(* IEC 61131-3 sources: Industry-PLC-LLM/data/PLCBEAD_repo/PLCBEAD_PLCEmbed-main/PLC-BEAD/Source/OpenPLCv2 (part 9) *)

(* ---- SRAMP.ST ---- *)
FUNCTION_BLOCK T_PLC_US_Block
	VAR_OUTPUT
		T_PLC_US :	UDINT;
	END_VAR

	VAR_EXTERNAL
		PLC_TICKS_PER_SEC :	INT;
		PLC_SYS_TICK_CNT :	DINT;
	END_VAR

	VAR
		debug :	BOOL;
		N :	INT;
		Offset :	UDINT;
		temp :	DWORD := DWORD#1;
		mode :	BOOL;
		faktor :	UDINT;
		init :	BOOL;
		v_plc_ticks_per_sec :	UDINT;
		base :	UDINT := UDINT#1000000;
	END_VAR

	IF init = FALSE THEN
		v_plc_ticks_per_sec := INT_TO_UDINT(PLC_TICKS_PER_SEC);
		IF v_plc_ticks_per_sec = UDINT#1024 THEN
			faktor := UDINT#1000;
			mode := FALSE;
		ELSIF v_plc_ticks_per_sec > UDINT#0 THEN
			IF v_plc_ticks_per_sec <= base THEN
				faktor := base / v_plc_ticks_per_sec;
				mode := FALSE;
			ELSE
				faktor := v_plc_ticks_per_sec / base;
				mode := TRUE;
			END_IF;
		ELSE
			faktor := UDINT#1;
		END_IF;
		init := TRUE;
	END_IF;

	IF mode THEN
		T_PLC_US := DINT_TO_UDINT(PLC_SYS_TICK_CNT) / faktor;
	ELSE
		T_PLC_US := DINT_TO_UDINT(PLC_SYS_TICK_CNT) * faktor;
	END_IF;

	IF debug THEN
		T_PLC_US := (DWORD_TO_UDINT(SHL(UDINT_TO_DWORD(T_PLC_US),N) OR SHL(temp,N)) - UDINT#1) + Offset;
	END_IF;
END_FUNCTION_BLOCK

FUNCTION_BLOCK TC_S_Block

	VAR_OUTPUT
		TC :	REAL;
	END_VAR

	VAR
		init :	BOOL;
		tx :	UDINT;
		last :	UDINT;
		T_PLC_US :	T_PLC_US_Block;
	END_VAR

	T_PLC_US();
	tx:= T_PLC_US.T_PLC_US;

	IF NOT init THEN
		init := TRUE;
		TC := 0.0;
	ELSE
		tc := UDINT_TO_REAL(tx - last) * 1.0E-6;
	END_IF;
	last := tx;

END_FUNCTION_BLOCK

FUNCTION_BLOCK SRAMP_Block

	VAR_INPUT
		X :	REAL;
		A_UP :	REAL;
		A_DN :	REAL;
		VU_MAX :	REAL;
		VD_MAX :	REAL;
		LIMIT_HIGH :	REAL;
		LIMIT_LOW :	REAL;
		RST :	BOOL;
	END_VAR

	VAR_OUTPUT
		Y :	REAL;
		V :	REAL;
	END_VAR

	VAR
		cycle_time :	TC_S_Block;
		init :	BOOL;
	END_VAR

	cycle_time();

	A_up := MAX(0.0,A_UP);
	A_dn := MIN(0.0,A_dn);
	VU_max := MAX(0.0,VU_max);
	VD_max := MIN(0.0,VD_MAX);

	IF rst OR NOT init THEN
		init := TRUE;
		Y := 0.0;
		V := 0.0;
	ELSIF X = Y THEN
		v := 0.0;
	ELSIF X > Y THEN
		v := MIN(v + A_UP * cycle_time.TC, vu_max);
		v := MIN(SQRT((Y-X) * 2.0 * A_DN), v);
		y := LIMIT(limit_low, y + MIN(v * cycle_time.TC, X-Y), limit_high);
	ELSIF X < Y THEN
		v := MAX(v + A_DN * cycle_time.TC, vd_max);
		v := MAX(-SQRT((Y-X) * 2.0 * A_UP), v);
		y := LIMIT(limit_low, y + MAX(v * cycle_time.TC, X-Y), limit_high);
	END_IF;

END_FUNCTION_BLOCK

PROGRAM program0
	VAR
		X :	REAL;
		A_UP :	REAL;
		A_DN :	REAL;
		VU_MAX :	REAL;
		VD_MAX :	REAL;
		LIMIT_HIGH :	REAL;
		LIMIT_LOW :	REAL;
		RST :	BOOL;
		Y :	REAL;
		V :	REAL;
		func_block : SRAMP_Block;
	END_VAR
		func_block.X  := X;
		func_block.A_UP  := A_UP;
		func_block.A_DN  := A_DN;
		func_block.VU_MAX  := VU_MAX;
		func_block.VD_MAX  := VD_MAX;
		func_block.LIMIT_HIGH  := LIMIT_HIGH;
		func_block.LIMIT_LOW  := LIMIT_LOW;
		func_block.RST  := RST;
		func_block();
		Y := func_block.Y;
		V := func_block.V;

END_PROGRAM

CONFIGURATION Config0

	VAR_GLOBAL
		PLC_TICKS_PER_SEC :	INT;
		PLC_SYS_TICK_CNT :	DINT;
	END_VAR

	RESOURCE Res0 ON PLC
		TASK task0(INTERVAL := T#20ms,PRIORITY := 0);
		PROGRAM instance0 WITH task0 : program0;
	END_RESOURCE

END_CONFIGURATION

(* ---- STACK_16.ST ---- *)
TYPE
  oscat_ardw_0_15             : ARRAY [0..15]   OF DWORD;
END_TYPE

FUNCTION_BLOCK STACK_16_Block

	VAR_INPUT
		DIN :	DWORD;
		E :	BOOL := TRUE;
		RD :	BOOL;
		WD :	BOOL;
		RST :	BOOL;
	END_VAR

	VAR_OUTPUT
		DOUT :	DWORD;
		EMPTY :	BOOL := TRUE;
		FULL :	BOOL;
	END_VAR

	VAR
		pt :	INT;
		stack :	oscat_ardw_0_15;
	END_VAR

	IF RST THEN
		pt := 0;
		EMPTY := TRUE;
		FULL := FALSE;
		Dout := DWORD#0;
	ELSIF E THEN
		IF NOT EMPTY AND RD THEN
			pt := pt - 1;
			Dout := stack[pt];
			EMPTY := pt = 0;
			FULL := FALSE;
		END_IF;
		IF NOT FULL AND WD THEN
			stack[pt] := Din;
			pt := pt + 1;
			FULL := pt > 15;
			EMPTY := FALSE;
		END_IF;
	END_IF;

END_FUNCTION_BLOCK

PROGRAM program0
	VAR
		DIN :	DWORD;
		E :	BOOL := TRUE;
		RD :	BOOL;
		WD :	BOOL;
		RST :	BOOL;
		DOUT :	DWORD;
		EMPTY :	BOOL := TRUE;
		FULL :	BOOL;
		func_block : STACK_16_Block;
	END_VAR
		func_block.DIN  := DIN;
		func_block.E  := E;
		func_block.RD  := RD;
		func_block.WD  := WD;
		func_block.RST  := RST;
		func_block();
		DOUT := func_block.DOUT;
		EMPTY := func_block.EMPTY;
		FULL := func_block.FULL;

END_PROGRAM

CONFIGURATION Config0

	RESOURCE Res0 ON PLC
		TASK task0(INTERVAL := T#20ms,PRIORITY := 0);
		PROGRAM instance0 WITH task0 : program0;
	END_RESOURCE

END_CONFIGURATION

(* ---- STACK_32.ST ---- *)
TYPE
  	oscat_ardw_0_31             : ARRAY [0..31]   OF DWORD;
END_TYPE

FUNCTION_BLOCK STACK_32_Block

	VAR_INPUT
		DIN :	DWORD;
		E :	BOOL := TRUE;
		RD :	BOOL;
		WD :	BOOL;
		RST :	BOOL;
	END_VAR

	VAR_OUTPUT
		DOUT :	DWORD;
		EMPTY :	BOOL := TRUE;
		FULL :	BOOL;
	END_VAR

	VAR
		pt :	INT;
		stack :	oscat_ardw_0_31;
	END_VAR

	IF RST THEN
		pt := 0;
		EMPTY := TRUE;
		FULL := FALSE;
		Dout := DWORD#0;
	ELSIF E THEN
		IF NOT EMPTY AND RD THEN
			(* read one element *)
			pt := pt - 1;
			Dout := stack[pt];
			EMPTY := pt = 0;
			FULL := FALSE;
		END_IF;
		IF NOT FULL AND WD THEN
			(* write one element *)
			stack[pt] := Din;
			pt := pt + 1;
			FULL := pt > 31;
			EMPTY := FALSE;
		END_IF;
	END_IF;

END_FUNCTION_BLOCK

PROGRAM program0
	VAR
		DIN :	DWORD;
		E :	BOOL := TRUE;
		RD :	BOOL;
		WD :	BOOL;
		RST :	BOOL;
		DOUT :	DWORD;
		EMPTY :	BOOL := TRUE;
		FULL :	BOOL;
		func_block : STACK_32_Block;
	END_VAR
		func_block.DIN  := DIN;
		func_block.E  := E;
		func_block.RD  := RD;
		func_block.WD  := WD;
		func_block.RST  := RST;
		func_block();
		DOUT := func_block.DOUT;
		EMPTY := func_block.EMPTY;
		FULL := func_block.FULL;

END_PROGRAM

CONFIGURATION Config0

	RESOURCE Res0 ON PLC
		TASK task0(INTERVAL := T#20ms,PRIORITY := 0);
		PROGRAM instance0 WITH task0 : program0;
	END_RESOURCE

END_CONFIGURATION

(* ---- STAIR2.ST ---- *)
FUNCTION FLOOR : INT
	VAR_INPUT
		x : REAL;
	END_VAR

	FLOOR := REAL_TO_INT(X);
	IF INT_TO_REAL(FLOOR) > X THEN
		floor := floor - 1;
	END_IF;
END_FUNCTION

FUNCTION_BLOCK STAIR2_Block

	VAR_INPUT
		X :	REAL;
		D :	REAL;
	END_VAR

	VAR_OUTPUT
		Y :	REAL;
	END_VAR

	IF D > 0.0 THEN
		IF X >= Y + D OR X <= Y - D THEN Y := INT_TO_REAL(FLOOR(X/D)) * D; END_IF;
	ELSE
		Y := X;
	END_IF;

END_FUNCTION_BLOCK

PROGRAM program0

	VAR
		X :	REAL;
		D :	REAL;
		Y :	REAL;
		func_block : STAIR2_Block;
	END_VAR
	func_block.X := X;
	func_block.D := D;
	func_block();
	Y := func_block.Y;

END_PROGRAM

CONFIGURATION Config0

	RESOURCE Res0 ON PLC
		TASK task0(INTERVAL := T#20ms,PRIORITY := 0);
		PROGRAM instance0 WITH task0 : program0;
	END_RESOURCE

END_CONFIGURATION

(* ---- STATUS_TO_ESR.ST ---- *)
TYPE
  oscat_esr_collect_data      : ARRAY [0..7]    OF BYTE;
END_TYPE

TYPE oscat_esr_data :
  STRUCT
	typ    : BYTE;
	adress : STRING;
	DS     : UDINT;
	TS     : TIME;
	data   : oscat_esr_collect_data;
  END_STRUCT;
END_TYPE

FUNCTION_BLOCK STATUS_TO_ESR_Block

	VAR_INPUT
		STATUS :	BYTE;
		ADRESS :	STRING;
		DT_IN :	UDINT;
		TS :	TIME;
	END_VAR

	VAR_OUTPUT
		STATUS_TO_ESR :	oscat_esr_data;
	END_VAR

	IF status < BYTE#100 THEN
		status_to_ESR.typ := BYTE#1;
	ELSIF status < BYTE#200 THEN
		status_to_ESR.typ := BYTE#2;
	ELSE
		status_to_ESR.typ := BYTE#3;
	END_IF;
	status_to_ESR.adress:= adress;
	status_to_ESR.DS := DT_in;
	status_to_ESR.TS := TS;
	status_to_ESR.data[0] := status;
END_FUNCTION_BLOCK

PROGRAM program0
	VAR
		STATUS :	BYTE;
		ADRESS :	STRING;
		DT_IN  :	UDINT;
		TS     :	TIME;
		STATUS_TO_ESR :	oscat_esr_data;

		func_block : STATUS_TO_ESR_Block;
	END_VAR
	func_block.STATUS := STATUS;
	func_block.ADRESS := ADRESS;
	func_block.DT_IN := DT_IN ;
	func_block.TS    := TS    ;

	func_block();
	STATUS_TO_ESR  := func_block.STATUS_TO_ESR;
END_PROGRAM

CONFIGURATION Config0
	RESOURCE Res0 ON PLC
		TASK task0(INTERVAL := T#20ms,PRIORITY := 0);
		PROGRAM instance0 WITH task0 : program0;
	END_RESOURCE
END_CONFIGURATION

(* ---- STORE_8.ST ---- *)
FUNCTION_BLOCK STORE_8_Block

	VAR_INPUT
		SET :	BOOL;
		D0 :	BOOL;
		D1 :	BOOL;
		D2 :	BOOL;
		D3 :	BOOL;
		D4 :	BOOL;
		D5 :	BOOL;
		D6 :	BOOL;
		D7 :	BOOL;
		CLR :	BOOL;
		RST :	BOOL;
	END_VAR

	VAR_OUTPUT
		Q0 :	BOOL;
		Q1 :	BOOL;
		Q2 :	BOOL;
		Q3 :	BOOL;
		Q4 :	BOOL;
		Q5 :	BOOL;
		Q6 :	BOOL;
		Q7 :	BOOL;
	END_VAR

	VAR
		edge :	BOOL;
	END_VAR

	IF rst OR set THEN
		q0 := NOT rst;
		q1 := q0;
		q2 := q0;
		q3 := q0;
		q4 := q0;
		q5 := q0;
		q6 := q0;
		q7 := q0;
	ELSE
		IF D0 THEN Q0 := TRUE; END_IF;
		IF D1 THEN Q1 := TRUE; END_IF;
		IF D2 THEN Q2 := TRUE; END_IF;
		IF D3 THEN Q3 := TRUE; END_IF;
		IF D4 THEN Q4 := TRUE; END_IF;
		IF D5 THEN Q5 := TRUE; END_IF;
		IF D6 THEN Q6 := TRUE; END_IF;
		IF D7 THEN Q7 := TRUE; END_IF;

		IF clr AND NOT edge THEN
			IF q0 THEN q0 := FALSE;
			ELSIF q1 THEN q1 := FALSE;
			ELSIF q2 THEN q2 := FALSE;
			ELSIF q3 THEN q3 := FALSE;
			ELSIF q4 THEN q4 := FALSE;
			ELSIF q5 THEN q5 := FALSE;
			ELSIF q6 THEN q6 := FALSE;
			ELSE q7 := FALSE;
			END_IF;
		END_IF;
		edge := clr;
	END_IF;

END_FUNCTION_BLOCK

PROGRAM program0
	VAR
		SET :	BOOL;
		D0 :	BOOL;
		D1 :	BOOL;
		D2 :	BOOL;
		D3 :	BOOL;
		D4 :	BOOL;
		D5 :	BOOL;
		D6 :	BOOL;
		D7 :	BOOL;
		CLR :	BOOL;
		RST :	BOOL;
		Q0 :	BOOL;
		Q1 :	BOOL;
		Q2 :	BOOL;
		Q3 :	BOOL;
		Q4 :	BOOL;
		Q5 :	BOOL;
		Q6 :	BOOL;
		Q7 :	BOOL;
		func_block : STORE_8_Block;
	END_VAR
	func_block.SET  := SET;
	func_block.D0  := D0;
	func_block.D1  := D1;
	func_block.D2  := D2;
	func_block.D3  := D3;
	func_block.D4  := D4;
	func_block.D5  := D5;
	func_block.D6  := D6;
	func_block.D7  := D7;
	func_block.CLR  := CLR;
	func_block.RST  := RST;
	func_block();
	Q0  := func_block.Q0;
	Q1  := func_block.Q1;
	Q2  := func_block.Q2;
	Q3  := func_block.Q3;
	Q4  := func_block.Q4;
	Q5  := func_block.Q5;
	Q6  := func_block.Q6;
	Q7  := func_block.Q7;
END_PROGRAM

CONFIGURATION Config0
	RESOURCE Res0 ON PLC
		TASK task0(INTERVAL := T#20ms,PRIORITY := 0);
		PROGRAM instance0 WITH task0 : program0;
	END_RESOURCE
END_CONFIGURATION

(* ---- STRING_TO_TOD.ST ---- *)
FUNCTION_BLOCK STRING_TO_TOD_Block

  VAR_INPUT
    _TOD :	STRING;
  END_VAR

  VAR_OUTPUT
    out_STRING_TO_TOD :	UDINT;
  END_VAR

  VAR
    pos :	INT;
    i :	INT;
    tmp :	STRING;
    tmp2 :	STRING;
  END_VAR

  out_STRING_TO_TOD := UDINT#0;
  i := LEN(_TOD);
  pos :=FIND(_TOD,'#');

  IF pos>0 AND i>pos THEN
    tmp := RIGHT(_TOD,LEN(_TOD)-pos);
    pos := FIND(tmp,':');
    IF pos>1 THEN
      tmp2 := LEFT(tmp,pos-1);
      tmp := RIGHT(tmp,LEN(tmp)-pos);
      out_STRING_TO_TOD := STRING_TO_UDINT(tmp2) * UDINT#3600000;

      pos :=FIND(tmp,':');
      IF pos>1 THEN
        tmp2 := LEFT(tmp,pos-1);
        tmp := RIGHT(tmp,LEN(tmp)-pos);
        out_STRING_TO_TOD := out_STRING_TO_TOD + STRING_TO_UDINT(tmp2) * UDINT#60000;

        out_STRING_TO_TOD := out_STRING_TO_TOD + STRING_TO_UDINT(tmp) * UDINT#1000;
      END_IF;
    END_IF;
  END_IF;

END_FUNCTION_BLOCK

PROGRAM program0
  VAR
    _TOD :	STRING;
  	out_STRING_TO_TOD :	UDINT;
    func_block : STRING_TO_TOD_Block;
  END_VAR
	func_block._TOD  := _TOD;
	func_block();
	out_STRING_TO_TOD  := func_block.out_STRING_TO_TOD;
END_PROGRAM

CONFIGURATION Config0
	RESOURCE Res0 ON PLC
		TASK task0(INTERVAL := T#20ms,PRIORITY := 0);
		PROGRAM instance0 WITH task0 : program0;
	END_RESOURCE
END_CONFIGURATION

(* ---- STRING_TO_URL.ST ---- *)
TYPE
  oscat_STRING250             : STRING;
  oscat_STRING32             : STRING;
  oscat_STRING80             : STRING;
  oscat_STRING160             : STRING;
  oscat_STRING40             : STRING;
  oscat_STRING10             : STRING;
  oscat_STRING20             : STRING;
END_TYPE

TYPE oscat_url :
    STRUCT
    PROTOCOL : oscat_STRING10;
    USER     : oscat_STRING32;
    PASSWORD : oscat_STRING32;
    DOMAIN   : oscat_STRING80;
    PORT     : WORD;
    PATH     : oscat_STRING80;
    QUERY    : oscat_STRING250;
    ANCHOR   : oscat_STRING40;
    HEADER   : oscat_STRING160;
    END_STRUCT;
END_TYPE

FUNCTION_BLOCK STRING_TO_URL_Block

	VAR_INPUT
		STR :	oscat_STRING250;
		DEFAULT_PROTOCOL :	oscat_STRING20 := 'http';
		DEFAULT_PATH :	oscat_STRING80 := '/';
	END_VAR

	VAR_OUTPUT
		STRING_TO_URL :	oscat_url;
	END_VAR

	VAR
		pos :	INT;
		pos2 :	INT;
		temp :	STRING;
		x :	oscat_STRING250;
	END_VAR

	IF EQ_STRING(STR,'') THEN
		RETURN;
	END_IF;

	pos := FIND(STR, '://');
	IF pos > 0 THEN
		STRING_TO_URL.PROTOCOL := LEFT(STR, pos - 1);
		x := RIGHT(STR, LEN(STR) - pos - 2);
	ELSE
		x := STR;
		STRING_TO_URL.PROTOCOL := DEFAULT_PROTOCOL;
	END_IF;

	pos := FIND(x, '@');
	IF pos > 0 THEN
		pos2 := FIND(x,':')+1;
		IF pos2 > 1 AND pos2 <= pos THEN
			STRING_TO_URL.USER := LEFT(x,pos2 - 2);
			STRING_TO_URL.PASSWORD := MID(x, pos - pos2, pos2);
		ELSE
			STRING_TO_URL.USER := LEFT(x, pos - 2);
			STRING_TO_URL.PASSWORD := '';
		END_IF;
		x := RIGHT(x, LEN(x) - pos);
	ELSE
		STRING_TO_URL.USER := '';
		STRING_TO_URL.PASSWORD := '';
	END_IF;

	pos := FIND(x, '#');
	IF pos > 0 THEN
		STRING_TO_URL.ANCHOR := RIGHT(x, LEN(x) - pos);
		x := LEFT(x, pos - 1);
	ELSE
		STRING_TO_URL.ANCHOR := '';
	END_IF;

	pos := FIND(x, '?');
	IF pos > 0 THEN
		STRING_TO_URL.QUERY := RIGHT(x, LEN(x) - pos);
		x := LEFT(x, pos - 1);
	ELSE
		STRING_TO_URL.QUERY := '';
	END_IF;

	pos := FIND(x, '/');
	IF pos > 0 THEN
		STRING_TO_URL.PATH := RIGHT(x, LEN(x) - pos + 1);
		x := LEFT(x, pos - 1);
	ELSE
		STRING_TO_URL.PATH := DEFAULT_PATH;
	END_IF;

	pos := FIND(x, ':');
	IF pos > 0 THEN
		temp := RIGHT(x, LEN(x) - pos);
		STRING_TO_URL.PORT := STRING_TO_WORD(temp);
		STRING_TO_URL.DOMAIN := LEFT(x, pos - 1);
	ELSE
		STRING_TO_URL.PORT := WORD#0;
		STRING_TO_URL.DOMAIN := x;
	END_IF;

END_FUNCTION_BLOCK

PROGRAM program0
	VAR
		STR :	oscat_STRING250;
		DEFAULT_PROTOCOL :	oscat_STRING20 := 'http';
		DEFAULT_PATH :	oscat_STRING80 := '/';
		STRING_TO_URL :	oscat_url;

		func_block : STRING_TO_URL_Block;
	END_VAR
	func_block.STR := STR;
	func_block.DEFAULT_PROTOCOL := DEFAULT_PROTOCOL;
	func_block.DEFAULT_PATH := DEFAULT_PATH;

	func_block();
  	STRING_TO_URL  := func_block.STRING_TO_URL;
END_PROGRAM

CONFIGURATION Config0
	RESOURCE Res0 ON PLC
		TASK task0(INTERVAL := T#20ms,PRIORITY := 0);
		PROGRAM instance0 WITH task0 : program0;
	END_RESOURCE
END_CONFIGURATION

(* ---- SUN_POS.ST ---- *)
FUNCTION FLOOR2 : DINT
	VAR_INPUT
		x : REAL;
	END_VAR

	FLOOR2 := REAL_TO_DINT(X);
	IF DINT_TO_REAL(FLOOR2) > X THEN
		FLOOR2 := FLOOR2 - DINT#1;
	END_IF;

END_FUNCTION

FUNCTION MODR:REAL

	VAR_INPUT
		IN :	REAL;
		DIVI :	REAL;
	END_VAR

	IF divi = 0.0 THEN
		MODR := 0.0;
	ELSE
		MODR := in - DINT_TO_REAL(FLOOR2(in / divi)) * divi;
	END_IF;

END_FUNCTION

FUNCTION RAD:REAL

	VAR_INPUT
		DEGG :	REAL;
	END_VAR

	RAD := MODR(0.0174532925199433 * DEGG , 6.283185307179586476);

END_FUNCTION

FUNCTION REFRACTION:REAL

	VAR_INPUT
		ELEV :	REAL;
	END_VAR

	VAR
		tmp :	REAL;
	END_VAR

	tmp := LIMIT(-1.9, elev, 80.0);
	REFRACTION := 0.0174532925199433 / TAN(0.0174532925199433 * (tmp + 10.3 / (tmp + 5.11)));

END_FUNCTION

FUNCTION TOD_TO_REAL2:REAL
	VAR_INPUT
		IN :	UDINT;
	END_VAR
	TOD_TO_REAL2 := UDINT_TO_REAL(IN);
END_FUNCTION

FUNCTION DEG:REAL

	VAR_INPUT
		X :	REAL;
	END_VAR

	DEG := MODR(57.29577951308232 * X, 360.0);
END_FUNCTION

FUNCTION DT_TO_TOD2:UDINT
	VAR_INPUT
		IN :	UDINT;
	END_VAR

	DT_TO_TOD2 := (IN MOD UDINT#86400) * UDINT#1000;
END_FUNCTION

FUNCTION_BLOCK SUN_POS

	VAR_INPUT
		LATITUDE :	REAL;
		LONGITUDE :	REAL;
		UTC :	UDINT;
	END_VAR

	VAR_OUTPUT
		B :	REAL;
		HR :	REAL;
	END_VAR

	VAR
		g :	REAL;
		a :	REAL;
		d :	REAL;
		h :	REAL;
		t1 :	REAL;
		n :	REAL;
		e :	REAL;
		c :	REAL;
		tau :	REAL;
		sin_d :	REAL;
		rlat :	REAL;
		sin_lat :	REAL;
		cos_lat :	REAL;
		cos_tau :	REAL;
		cos_d :	REAL;
		MATH_PI :	REAL := 3.14159265358979323846264338327950288;
		MATH_PI2 :	REAL := 6.28318530717958647692528676655900576;
	END_VAR

	n := UDINT_TO_REAL(UTC - UDINT#946728000) * 0.000011574074074074;
	g :=MODR(6.240040768 + 0.01720197 * n, MATH_PI2);
	d := MODR(4.89495042 + 0.017202792 * n, MATH_PI2) + 0.033423055 * SIN(g) + 0.000349066 * SIN(2.0*g);
	e := 0.409087723 - 0.000000006981317008 * n;
	cos_d := COS(d);
	sin_d := SIN(d);
	a := ATAN(COS(e) * sin_d / cos_d);
	IF cos_d < 0.0 THEN a := a + MATH_PI; END_IF;
	c := ASIN(SIN(e) * sin_d);

	(* also here we must be very careful utc is from 1.1.1970 for step7 the formula must change *)
	tau := RAD(MODR(6.697376 + (n - 0.25) * 0.0657098245037645 + TOD_TO_REAL2(DT_TO_TOD2(utc)) * 0.0000002785383333, 24.0) * 15.0 + longitude) - a;
	rlat := RAD(latitude);
	sin_lat := SIN(rlat);
	cos_lat := COS(rlat);
	cos_tau := COS(tau);
	t1 := cos_tau * sin_lat - TAN(c) * cos_lat;
	B := ATAN(SIN(tau) / t1);
	IF t1 < 0.0 THEN B := B + MATH_PI2; ELSE B := B + MATH_PI; END_IF;
	B := DEG(MODR(B, MATH_PI2));
	h := DEG(ASIN(COS(C) * cos_tau * cos_lat +SIN(c) * sin_lat));
	IF h > 180.0 THEN h := h - 360.0; END_IF;
	(* consider refraction *)
	HR := h + REFRACTION(h);
END_FUNCTION_BLOCK

PROGRAM program0
  VAR
	LATITUDE :	REAL;
	LONGITUDE :	REAL;
	UTC :	UDINT;
	B :	REAL;
	HR :	REAL;
	func_block : SUN_POS;
  END_VAR
	func_block.LATITUDE  :=LATITUDE ;
	func_block.LONGITUDE  :=LONGITUDE ;
	func_block.UTC  :=UTC ;
	func_block();
	B := func_block.B;
	HR := func_block.HR;
END_PROGRAM

CONFIGURATION Config0
	RESOURCE Res0 ON PLC
		TASK task0(INTERVAL := T#20ms,PRIORITY := 0);
		PROGRAM instance0 WITH task0 : program0;
	END_RESOURCE
END_CONFIGURATION

(* ---- SW_RECONFIG.ST ---- *)
FUNCTION_BLOCK SW_RECONFIG_Block

	VAR_INPUT
		IN :	BOOL;
		TD :	TIME;
		TR :	TIME;
	END_VAR

	VAR_OUTPUT
		Q :	BOOL;
	END_VAR

	VAR
		T1 :	TON;
		T2 :	TON;
		INV :	BOOL;
	END_VAR

	t1(in := IN, PT := TD);

	IF tr > t#0s THEN
		Q := t1.Q XOR inv;
		T2(in := Q, pt := TR);
		IF T2.Q THEN INV := NOT INV; END_IF;
	ELSE
		Q := t1.Q;
	END_IF;

END_FUNCTION_BLOCK

PROGRAM program0
	VAR
		IN :	BOOL;
		TD :	TIME;
		TR :	TIME;
		Q :	BOOL;

		func_block : SW_RECONFIG_Block;
	END_VAR
	func_block.IN := IN;
	func_block.TD := TD;
	func_block.TR := TR ;

	func_block();
	Q  := func_block.Q;

END_PROGRAM

CONFIGURATION Config0
	RESOURCE Res0 ON PLC
		TASK task0(INTERVAL := T#20ms,PRIORITY := 0);
		PROGRAM instance0 WITH task0 : program0;
	END_RESOURCE
END_CONFIGURATION

(* ---- SWITCH_I.ST ---- *)
FUNCTION UDINT_TO_TIME2:TIME

	VAR_INPUT
		IN :	UDINT;
	END_VAR

	UDINT_TO_TIME2 := DINT_TO_TIME(UDINT_TO_DINT(IN));

END_FUNCTION

FUNCTION_BLOCK T_PLC_MS_block
	VAR_OUTPUT
		T_PLC_MS :	UDINT;
	END_VAR

	VAR_EXTERNAL
		PLC_TICKS_PER_SEC :	INT;
		PLC_SYS_TICK_CNT :	DINT;
	END_VAR

	VAR
		debug :	BOOL;(*Debug-Mode ON / OFF*)
		N :	INT;(*Debug-Faktor*)
		Offset :	UDINT;(*Debug-Offset*)
		temp :	DWORD := DWORD#1;(*Debug-Offset*)
		mode :	BOOL;(*modus*)
		faktor :	UDINT;(*Systemtakt-Faktor*)
		init :	BOOL;
		v_plc_ticks_per_sec :	UDINT;
		base :	UDINT := UDINT#1000;
	END_VAR

	IF init = FALSE THEN
		v_plc_ticks_per_sec := INT_TO_UDINT(PLC_TICKS_PER_SEC);
		IF v_plc_ticks_per_sec = UDINT#1024 THEN
			faktor := UDINT#1;
			mode := FALSE;
		ELSIF v_plc_ticks_per_sec > UDINT#0 THEN
			IF v_plc_ticks_per_sec <= base THEN
				faktor := base / v_plc_ticks_per_sec;
				mode := FALSE;
			ELSE
				faktor := v_plc_ticks_per_sec / base;
				mode := TRUE;
			END_IF;
		ELSE
			faktor := UDINT#1;
		END_IF;
		init := TRUE;
	END_IF;

	IF mode THEN
		T_PLC_MS := DINT_TO_UDINT(PLC_SYS_TICK_CNT) / faktor;
	ELSE
		T_PLC_MS := DINT_TO_UDINT(PLC_SYS_TICK_CNT) * faktor;
	END_IF;

	IF debug THEN
		T_PLC_MS := (DWORD_TO_UDINT(SHL(UDINT_TO_DWORD(T_PLC_MS),N) OR SHL(temp,N)) - UDINT#1) + Offset;
	END_IF;

END_FUNCTION_BLOCK

FUNCTION_BLOCK SWITCH_I_Block

	VAR_INPUT
		SET :	BOOL;
		IN :	BOOL;
		RST :	BOOL;
		T_DEBOUNCE :	TIME := T#10ms;
		T_RECONFIG :	TIME := T#1s;
		T_ON_MAX :	TIME := T#0h;
	END_VAR

	VAR_OUTPUT
		Q :	BOOL := FALSE;
	END_VAR

	VAR
		state :	BYTE := BYTE#0;
		edge :	BOOL := FALSE;
		_r_edge :	BOOL := FALSE;
		T_on :	TIME;
		tx :	TIME;
		T_PLC_MS :	T_PLC_MS_Block;
	END_VAR

	T_PLC_MS();
	tx:= UDINT_TO_TIME(T_PLC_MS.T_PLC_MS);

	IF set AND NOT rst THEN
		Q := TRUE;
		T_on := tx;
	ELSIF rst THEN
		Q := FALSE;
	ELSIF (in XOR edge) AND NOT (state = BYTE#1) THEN
		state := BYTE#1;
		T_on := Tx;
	ELSIF (state = BYTE#1) AND (Tx - t_debounce >= T_on) THEN
		state := BYTE#2;
		IF _r_edge XOR in THEN Q := NOT Q;
	END_IF;
	ELSIF state = BYTE#2 AND Tx - t_reconfig >= T_on THEN
		_r_edge := in;
	END_IF;
	IF Q AND T_on_max > t#0ms AND Tx >= T_on + T_on_max THEN
		Q := FALSE;
	END_IF;
	edge := in;

END_FUNCTION_BLOCK

PROGRAM program0
	VAR
		SET :	BOOL;
		IN :	BOOL;
		RST :	BOOL;
		T_DEBOUNCE :	TIME := T#10ms;
		T_RECONFIG :	TIME := T#1s;
		T_ON_MAX :	TIME := T#0h;
		Q :	BOOL := FALSE;

		func_block : SWITCH_I_Block;
	END_VAR
	func_block.SET := SET;
	func_block.IN := IN;
	func_block.RST := RST ;
	func_block.T_DEBOUNCE := T_DEBOUNCE ;
	func_block.T_RECONFIG := T_RECONFIG ;
	func_block.T_ON_MAX := T_ON_MAX ;

	func_block();
	Q  := func_block.Q;
END_PROGRAM

CONFIGURATION Config0
	VAR_GLOBAL
		PLC_TICKS_PER_SEC :	INT;
		PLC_SYS_TICK_CNT :	DINT;
	END_VAR
  	RESOURCE Res0 ON PLC
    	TASK task0(INTERVAL := T#20ms,PRIORITY := 0);
    	PROGRAM instance0 WITH task0 : program0;
  	END_RESOURCE
END_CONFIGURATION

(* ---- SWITCH_X.ST ---- *)
FUNCTION_BLOCK SWITCH_X_Block

	VAR_INPUT
		IN1 :	BOOL;
		IN2 :	BOOL;
		IN3 :	BOOL;
		IN4 :	BOOL;
		IN5 :	BOOL;
		IN6 :	BOOL;
		T_DEBOUNCE :	TIME := T#50ms;
	END_VAR

	VAR_OUTPUT
		Q1 :	BOOL;
		Q2 :	BOOL;
		Q3 :	BOOL;
		Q4 :	BOOL;
		Q5 :	BOOL;
		Q6 :	BOOL;
		Q31 :	BOOL;
		Q41 :	BOOL;
		Q51 :	BOOL;
		Q61 :	BOOL;
		Q32 :	BOOL;
		Q42 :	BOOL;
		Q52 :	BOOL;
		Q62 :	BOOL;
	END_VAR

	VAR
		INIT :	BOOL;
		T1 :	TOF;
		T2 :	TOF;
		T3 :	TOF;
		T4 :	TOF;
		T5 :	TOF;
		T6 :	TOF;
		tx :	TIME;
		x1 :	BOOL;
		x2 :	BOOL;
		E1 :	BOOL;
		E2 :	BOOL;
	END_VAR

	IF NOT init THEN
		init := TRUE;
		IF t_debounce < t#50ms THEN tx := t#50ms; ELSE tx := t_debounce; END_IF;
		T1(PT := Tx);
		T2(PT := Tx);
		T3(PT := Tx);
		T4(PT := Tx);
		T5(PT := Tx);
		T6(PT := Tx);
	ELSE
		Q1 := FALSE;
		Q2 := FALSE;
		Q3 := FALSE;
		Q4 := FALSE;
		Q5 := FALSE;
		Q6 := FALSE;
		Q31 := FALSE;
		Q41 := FALSE;
		Q51 := FALSE;
		Q61 := FALSE;
		Q32 := FALSE;
		Q42 := FALSE;
		Q52 := FALSE;
		Q62 := FALSE;
	END_IF;

		T1(IN := IN1);
		T2(IN := IN2);
		T3(IN := IN3);
		T4(IN := IN4);
		T5(IN := IN5);
		T6(IN := IN6);

	IF t1.Q AND NOT E1 THEN X1 := TRUE; END_IF;
	IF t2.Q AND NOT E2 THEN X2 := TRUE; END_IF;

	IF t1.Q THEN
		IF t3.q THEN
			q31 := TRUE;
			X1 := FALSE;
		ELSIF t4.q THEN
			q41 := TRUE;
			X1 := FALSE;
		ELSIF t5.q THEN
			q51 := TRUE;
			X1 := FALSE;
		ELSIF t6.q THEN
			q61 := TRUE;
			X1 := FALSE;
		END_IF;
	ELSIF t2.Q THEN
		IF t3.q THEN
			q32 := TRUE;
			X2 := FALSE;
		ELSIF t4.q THEN
			q42 := TRUE;
			X2 := FALSE;
		ELSIF t5.q THEN
			q52 := TRUE;
			X2 := FALSE;
		ELSIF t6.q THEN
			q62 := TRUE;
			X2 := FALSE;
		END_IF;
	ELSIF NOT T1.Q AND E1 AND X1 THEN
		Q1 := TRUE;
		X1 := FALSE;
	ELSIF NOT T2.Q AND E2 AND X2 THEN
		Q2 := TRUE;
		X2 := FALSE;
	ELSIF T3.Q THEN
		Q3 := TRUE;
	ELSIF T4.Q THEN
		Q4 := TRUE;
	ELSIF T5.Q THEN
		Q5 := TRUE;
	ELSIF T6.Q THEN
		Q6 := TRUE;
	END_IF;

	E1 := T1.Q;
	E2 := T2.Q;
END_FUNCTION_BLOCK

PROGRAM program0
	VAR
		IN1 :	BOOL;
		IN2 :	BOOL;
		IN3 :	BOOL;
		IN4 :	BOOL;
		IN5 :	BOOL;
		IN6 :	BOOL;
		T_DEBOUNCE :	TIME := T#50ms;
		Q1 :	BOOL;
		Q2 :	BOOL;
		Q3 :	BOOL;
		Q4 :	BOOL;
		Q5 :	BOOL;
		Q6 :	BOOL;
		Q31 :	BOOL;
		Q41 :	BOOL;
		Q51 :	BOOL;
		Q61 :	BOOL;
		Q32 :	BOOL;
		Q42 :	BOOL;
		Q52 :	BOOL;
		Q62 :	BOOL;

		func_block : SWITCH_X_Block;
	END_VAR
	func_block.IN1 := IN1;
	func_block.IN2 := IN2;
	func_block.IN3 := IN3 ;
	func_block.IN4 := IN4;
	func_block.IN5 := IN5;
	func_block.IN6 := IN6 ;
	func_block.T_DEBOUNCE := T_DEBOUNCE;

	func_block();
	Q1  := func_block.Q1;
	Q2  := func_block.Q2;
	Q3  := func_block.Q3;
	Q4  := func_block.Q4;
	Q5  := func_block.Q5;
	Q6  := func_block.Q6;
	Q31  := func_block.Q31;
	Q41  := func_block.Q41;
	Q51  := func_block.Q51;
	Q61  := func_block.Q61;
	Q32  := func_block.Q32;
	Q42  := func_block.Q42;
	Q52  := func_block.Q52;
	Q62  := func_block.Q62;

END_PROGRAM

CONFIGURATION Config0
	RESOURCE Res0 ON PLC
		TASK task0(INTERVAL := T#20ms,PRIORITY := 0);
		PROGRAM instance0 WITH task0 : program0;
	END_RESOURCE
END_CONFIGURATION

(* ---- T_AVG24.ST ---- *)
TYPE
  oscat_T_AVG24         	  : ARRAY [0..47]   OF INT;
END_TYPE

FUNCTION_BLOCK T_PLC_MS_block
	VAR_OUTPUT
		T_PLC_MS :	UDINT;
	END_VAR

	VAR_EXTERNAL
		PLC_TICKS_PER_SEC :	INT;
		PLC_SYS_TICK_CNT :	DINT;
	END_VAR

	VAR
		debug :	BOOL;(*Debug-Mode ON / OFF*)
		N :	INT;(*Debug-Faktor*)
		Offset :	UDINT;(*Debug-Offset*)
		temp :	DWORD := DWORD#1;(*Debug-Offset*)
		mode :	BOOL;(*modus*)
		faktor :	UDINT;(*Systemtakt-Faktor*)
		init :	BOOL;
		v_plc_ticks_per_sec :	UDINT;
		base :	UDINT := UDINT#1000;
	END_VAR

	IF init = FALSE THEN
		v_plc_ticks_per_sec := INT_TO_UDINT(PLC_TICKS_PER_SEC);
		IF v_plc_ticks_per_sec = UDINT#1024 THEN
			faktor := UDINT#1;
			mode := FALSE;
		ELSIF v_plc_ticks_per_sec > UDINT#0 THEN
			IF v_plc_ticks_per_sec <= base THEN
				faktor := base / v_plc_ticks_per_sec;
				mode := FALSE;
			ELSE
				faktor := v_plc_ticks_per_sec / base;
				mode := TRUE;
			END_IF;
		ELSE
			faktor := UDINT#1;
		END_IF;
		init := TRUE;
	END_IF;

	IF mode THEN
		T_PLC_MS := DINT_TO_UDINT(PLC_SYS_TICK_CNT) / faktor;
	ELSE
		T_PLC_MS := DINT_TO_UDINT(PLC_SYS_TICK_CNT) * faktor;
	END_IF;

	IF debug THEN
		T_PLC_MS := (DWORD_TO_UDINT(SHL(UDINT_TO_DWORD(T_PLC_MS),N) OR SHL(temp,N)) - UDINT#1) + Offset;
	END_IF;

END_FUNCTION_BLOCK

FUNCTION_BLOCK FILTER_I_Block
	VAR_INPUT
		X :	INT;
		T :	TIME;
	END_VAR

	VAR_OUTPUT
		Y :	INT;
	END_VAR

	VAR
		Yi :	DINT;
		last :	UDINT;
		tx :	UDINT;
		init :	BOOL;
		T_PLC_MS :	T_PLC_MS_block;
	END_VAR

	T_PLC_MS();
	tx:= T_PLC_MS.T_PLC_MS;

	IF NOT init OR T = t#0s THEN
		init := TRUE;
		Yi := INT_TO_DINT(X) * DINT#1000;
	ELSE
		Yi := Yi + INT_TO_DINT(X - Y) * UDINT_TO_DINT(tx - last) * DINT#1000 / TIME_TO_DINT(T);
	END_IF;
	last := tx;
	Y := DINT_TO_INT(yi / DINT#1000);

END_FUNCTION_BLOCK

FUNCTION TIME_TO_UDINT2:UDINT
	VAR_INPUT
		X :	TIME;
	END_VAR

	TIME_TO_UDINT2 := DINT_TO_UDINT(TIME_TO_DINT(X));
END_FUNCTION

FUNCTION INC1:INT

	VAR_INPUT
		X :	INT;
		N :	INT;
	END_VAR

	IF X >= N - 1 THEN
		INC1 := 0;
	ELSE
		INC1 := X + 1;
	END_IF;
END_FUNCTION

FUNCTION_BLOCK T_AVG24_Block

	VAR_INPUT
		TS :	INT;
		DTI :	UDINT;
		RST :	BOOL;
		T_FILTER :	TIME := T#10m;
		SCALE :	REAL := 1.0;
		OFS :	REAL;
	END_VAR

	VAR_OUTPUT
		TA :	REAL;
		_TP :	BOOL;
	END_VAR

	VAR_IN_OUT
		T24 :	REAL;
		T24_MAX :	REAL;
		T24_MIN :	REAL;
	END_VAR

	VAR
		samples :	oscat_T_AVG24;
		pos :	INT;
		init :	BOOL;
		sum :	DINT;
		last :	UDINT;
		tmp_maxxx :	INT;
		tmp_min :	INT;
		i :	INT;
		ft1 :	FILTER_I_Block;
	END_VAR

	ft1(X := TS, T := T_FILTER);

	IF rst OR NOT init THEN
		init := TRUE;
		IF T24 = -1000.0 THEN t24 := INT_TO_REAL(ft1.Y) * 0.1; END_IF;
		FOR pos := 0 TO 47 DO
			samples[pos] := REAL_TO_INT(T24 * 10.0);
		END_FOR;
		pos := 0;
		sum := INT_TO_DINT(samples[0]) * DINT#48;
		TA := (INT_TO_REAL(ft1.Y) * 0.1 + OFS) * SCALE;
		T24 := (DINT_TO_REAL(sum) * 0.00208333333333 + OFS) * SCALE;
		_TP := TRUE;
	ELSIF (dti / UDINT#60 MOD UDINT#30) = UDINT#0 AND DTI > last THEN
		last := DTI + TIME_TO_UDINT2(T#1m);
		sum := sum - INT_TO_DINT(samples[pos]);
		samples[pos] := ft1.Y;
		sum := sum + INT_TO_DINT(samples[pos]);
		pos := INC1(pos, 48);
		TA := (INT_TO_REAL(ft1.Y) * 0.1 + OFS) * SCALE;
		T24 := (DINT_TO_REAL(sum) * 0.00208333333333 + OFS) * SCALE;
		tmp_maxxx := -32000;
		tmp_min := 32000;
		FOR i := 0 TO 47 DO
			tmp_maxxx := MAX(tmp_maxxx, samples[i]);
			tmp_min := MIN(tmp_min, samples[i]);
		END_FOR;
		T24_MAX := (INT_TO_REAL(tmp_maxxx) * 0.1 + OFS) * SCALE;
		T24_MIN := (INT_TO_REAL(tmp_min) * 0.1 + OFS) * SCALE;
		_TP := TRUE;
	ELSE
		_TP := FALSE;
	END_IF;

END_FUNCTION_BLOCK

PROGRAM program0
	VAR
		TS :	INT;
		DTI :	UDINT;
		RST :	BOOL;
		T_FILTER :	TIME := T#10m;
		SCALE :	REAL := 1.0;
		OFS :	REAL;
		TA :	REAL;
		_TP :	BOOL;

		func_block : T_AVG24_Block;
	END_VAR
	func_block.TS := TS;
	func_block.DTI := DTI;
	func_block.RST := RST ;
	func_block.T_FILTER := T_FILTER;
	func_block.SCALE := SCALE;
	func_block.OFS := OFS ;

	func_block();
	TA  := func_block.TA;
	_TP  := func_block._TP;

END_PROGRAM

CONFIGURATION Config0
	VAR_GLOBAL
		PLC_TICKS_PER_SEC :	INT;
		PLC_SYS_TICK_CNT :	DINT;
	END_VAR
  	RESOURCE Res0 ON PLC
    	TASK task0(INTERVAL := T#20ms,PRIORITY := 0);
    	PROGRAM instance0 WITH task0 : program0;
  	END_RESOURCE
END_CONFIGURATION

(* ---- T_PLC_MS.ST ---- *)
FUNCTION_BLOCK T_PLC_MS_block

	VAR_OUTPUT
		T_PLC_MS :	UDINT;
	END_VAR

	VAR_EXTERNAL
		PLC_TICKS_PER_SEC :	INT;
		PLC_SYS_TICK_CNT :	DINT;
	END_VAR

	VAR
		debug :	BOOL;(*Debug-Mode ON / OFF*)
		N :	INT;(*Debug-Faktor*)
		Offset :	UDINT;(*Debug-Offset*)
		temp :	DWORD := DWORD#1;(*Debug-Offset*)
		mode :	BOOL;(*modus*)
		faktor :	UDINT;(*Systemtakt-Faktor*)
		init :	BOOL;
		v_plc_ticks_per_sec :	UDINT;
		base :	UDINT := UDINT#1000;
	END_VAR

	IF init = FALSE THEN
		v_plc_ticks_per_sec := INT_TO_UDINT(PLC_TICKS_PER_SEC);
		IF v_plc_ticks_per_sec = UDINT#1024 THEN
			faktor := UDINT#1;
			mode := FALSE;
		ELSIF v_plc_ticks_per_sec > UDINT#0 THEN
			IF v_plc_ticks_per_sec <= base THEN
				faktor := base / v_plc_ticks_per_sec;
				mode := FALSE;
			ELSE
				faktor := v_plc_ticks_per_sec / base;
				mode := TRUE;
			END_IF;
		ELSE
			faktor := UDINT#1;
		END_IF;
		init := TRUE;
	END_IF;

	IF mode THEN
		T_PLC_MS := DINT_TO_UDINT(PLC_SYS_TICK_CNT) / faktor;
	ELSE
		T_PLC_MS := DINT_TO_UDINT(PLC_SYS_TICK_CNT) * faktor;
	END_IF;

	IF debug THEN
		T_PLC_MS := (DWORD_TO_UDINT(SHL(UDINT_TO_DWORD(T_PLC_MS),N) OR SHL(temp,N)) - UDINT#1) + Offset;
	END_IF;

END_FUNCTION_BLOCK

PROGRAM program0

	VAR
		LocalOUT  : UDINT;
		func_block : T_PLC_MS_block;
  	END_VAR

	func_block();
	LocalOUT := func_block.T_PLC_MS;

END_PROGRAM

CONFIGURATION Config0

	VAR_GLOBAL
		PLC_TICKS_PER_SEC :	INT;
		PLC_SYS_TICK_CNT :	DINT;
	END_VAR

  	RESOURCE Res0 ON PLC
    	TASK task0(INTERVAL := T#20ms,PRIORITY := 0);
    	PROGRAM instance0 WITH task0 : program0;
  	END_RESOURCE

END_CONFIGURATION

(* ---- T_PLC_US.ST ---- *)
FUNCTION_BLOCK T_PLC_US_Block

	VAR_OUTPUT
		T_PLC_US :	UDINT;
	END_VAR

	VAR_EXTERNAL
		PLC_TICKS_PER_SEC :	INT;
		PLC_SYS_TICK_CNT :	DINT;
	END_VAR

	VAR
		debug :	BOOL;
		N :	INT;
		Offset :	UDINT;
		temp :	DWORD := DWORD#1;
		mode :	BOOL;
		faktor :	UDINT;
		init :	BOOL;
		v_plc_ticks_per_sec :	UDINT;
		base :	UDINT := UDINT#1000000;
	END_VAR

	IF init = FALSE THEN
		v_plc_ticks_per_sec := INT_TO_UDINT(PLC_TICKS_PER_SEC);
		IF v_plc_ticks_per_sec = UDINT#1024 THEN
			faktor := UDINT#1000;
			mode := FALSE;
		ELSIF v_plc_ticks_per_sec > UDINT#0 THEN
			IF v_plc_ticks_per_sec <= base THEN
				faktor := base / v_plc_ticks_per_sec;
				mode := FALSE;
			ELSE
				faktor := v_plc_ticks_per_sec / base;
				mode := TRUE;
			END_IF;
		ELSE
			faktor := UDINT#1;
		END_IF;
		init := TRUE;
	END_IF;

	IF mode THEN
		T_PLC_US := DINT_TO_UDINT(PLC_SYS_TICK_CNT) / faktor;
	ELSE
		T_PLC_US := DINT_TO_UDINT(PLC_SYS_TICK_CNT) * faktor;
	END_IF;

	IF debug THEN
		T_PLC_US := (DWORD_TO_UDINT(SHL(UDINT_TO_DWORD(T_PLC_US),N) OR SHL(temp,N)) - UDINT#1) + Offset;
	END_IF;

END_FUNCTION_BLOCK

PROGRAM program0

	VAR
		T_PLC_US  : UDINT;
		func_block : T_PLC_US_Block;
	END_VAR
		func_block();
		T_PLC_US := func_block.T_PLC_US;

END_PROGRAM

CONFIGURATION Config0

	VAR_GLOBAL
		PLC_TICKS_PER_SEC :	INT;
		PLC_SYS_TICK_CNT :	DINT;
	END_VAR

	RESOURCE Res0 ON PLC
		TASK task0(INTERVAL := T#20ms,PRIORITY := 0);
		PROGRAM instance0 WITH task0 : program0;
	END_RESOURCE

END_CONFIGURATION

(* ---- TANK_LEVEL.ST ---- *)
FUNCTION_BLOCK TONOF

	VAR_INPUT
		IN :	BOOL;
		T_ON :	TIME;
		T_OFF :	TIME;
	END_VAR

	VAR_OUTPUT
		Q :	BOOL;
	END_VAR

	VAR
		X :	TON;
		old :	BOOL;
		mode :	BOOL;
	END_VAR

	IF IN XOR old THEN
	X(IN := FALSE, PT := SEL_TIME(IN,T_OFF,T_ON));
	mode := IN;
	old := IN;
	END_IF;
	X(IN := TRUE);
	IF X.Q THEN Q := mode;END_IF;

END_FUNCTION_BLOCK

FUNCTION UDINT_TO_TIME2:TIME

	VAR_INPUT
		IN :	UDINT;
	END_VAR

	UDINT_TO_TIME2 := DINT_TO_TIME(UDINT_TO_DINT(IN));

END_FUNCTION

FUNCTION_BLOCK T_PLC_MS_block
	VAR_OUTPUT
		T_PLC_MS :	UDINT;
	END_VAR

	VAR_EXTERNAL
		PLC_TICKS_PER_SEC :	INT;
		PLC_SYS_TICK_CNT :	DINT;
	END_VAR

	VAR
		debug :	BOOL;(*Debug-Mode ON / OFF*)
		N :	INT;(*Debug-Faktor*)
		Offset :	UDINT;(*Debug-Offset*)
		temp :	DWORD := DWORD#1;(*Debug-Offset*)
		mode :	BOOL;(*modus*)
		faktor :	UDINT;(*Systemtakt-Faktor*)
		init :	BOOL;
		v_plc_ticks_per_sec :	UDINT;
		base :	UDINT := UDINT#1000;
	END_VAR

	IF init = FALSE THEN
		v_plc_ticks_per_sec := INT_TO_UDINT(PLC_TICKS_PER_SEC);
		IF v_plc_ticks_per_sec = UDINT#1024 THEN
			faktor := UDINT#1;
			mode := FALSE;
		ELSIF v_plc_ticks_per_sec > UDINT#0 THEN
			IF v_plc_ticks_per_sec <= base THEN
				faktor := base / v_plc_ticks_per_sec;
				mode := FALSE;
			ELSE
				faktor := v_plc_ticks_per_sec / base;
				mode := TRUE;
			END_IF;
		ELSE
			faktor := UDINT#1;
		END_IF;
		init := TRUE;
	END_IF;

	IF mode THEN
		T_PLC_MS := DINT_TO_UDINT(PLC_SYS_TICK_CNT) / faktor;
	ELSE
		T_PLC_MS := DINT_TO_UDINT(PLC_SYS_TICK_CNT) * faktor;
	END_IF;

	IF debug THEN
		T_PLC_MS := (DWORD_TO_UDINT(SHL(UDINT_TO_DWORD(T_PLC_MS),N) OR SHL(temp,N)) - UDINT#1) + Offset;
	END_IF;
END_FUNCTION_BLOCK

FUNCTION TIME_TO_UDINT2:UDINT
	VAR_INPUT
		X :	TIME;
	END_VAR

	TIME_TO_UDINT2 := DINT_TO_UDINT(TIME_TO_DINT(X));
END_FUNCTION

FUNCTION_BLOCK ACTUATOR_COIL_Block

	VAR_INPUT
		IN :	BOOL;
		SELF_ACT_CYCLE :	TIME := T#10d;
		SELF_ACT_TIME :	TIME := T#1s;
	END_VAR

	VAR_OUTPUT
		OUT :	BOOL;
		STATUS :	BYTE;
	END_VAR

	VAR
		last :	UDINT;
		init :	BOOL;
		tx :	UDINT;
		now :	UDINT;
		T_PLC_MS :	T_PLC_MS_Block;
	END_VAR

	T_PLC_MS();
	now := T_PLC_MS.T_PLC_MS;

	IF NOT init THEN
		last := now;
		init := TRUE;
	ELSIF IN THEN
		OUT := TRUE;
		STATUS := BYTE#101;
		LAST := now;
	ELSE
		OUT := FALSE;
		STATUS := BYTE#100;
		tx := now - last;
		IF (self_act_cycle > T#0s) AND (tx >= TIME_TO_UDINT2(self_act_cycle)) THEN
			OUT := TRUE;
			STATUS := BYTE#102;
			IF tx >= TIME_TO_UDINT2(self_act_cycle + self_act_time) THEN
				last := now;
				OUT := FALSE;
				STATUS := BYTE#100;
			END_IF;
		END_IF;
	END_IF;

END_FUNCTION_BLOCK

FUNCTION_BLOCK TANK_LEVEL_Block

	VAR_INPUT
		LEVEL :	BOOL;
		LEAK :	BOOL;
		ACLR :	BOOL;
		MAX_VALVE_TIME :	TIME;
		LEVEL_DELAY_TIME :	TIME;
	END_VAR

	VAR_OUTPUT
		VALVE :	BOOL;
		ALARM :	BOOL;
		STATUS :	BYTE;
	END_VAR

	VAR
		cx :	ACTUATOR_COIL_Block;
		tn :	TON;
		tl :	TONOF;
		open :	BOOL;
	END_VAR

	tl(in := level, T_ON := level_delay_time, T_OFF := level_delay_time);
	open := tl.Q;

	IF ALARM THEN
		IF ACLR THEN
			ALARM := FALSE;
			STATUS := BYTE#101;
			cx(in := FALSE);
		END_IF;
		RETURN;
	ELSIF LEAK THEN
		cx(in := FALSE);
		ALARM := TRUE;
		STATUS := BYTE#1;
	ELSIF open THEN
		cx(in := TRUE);
		STATUS := BYTE#102;
	ELSE
		cx(in := FALSE);
		STATUS := BYTE#100;
	END_IF;

	tn(in := cx.out AND (MAX_VALVE_TIME > T#0s), PT := MAX_VALVE_TIME);
	IF tn.Q THEN
		ALARM := TRUE;
		STATUS := BYTE#2;
		cx(in := FALSE);
	END_IF;

	VALVE := cx.out;
END_FUNCTION_BLOCK

PROGRAM program0
	VAR
		LEVEL :	BOOL;
		LEAK :	BOOL;
		ACLR :	BOOL;
		MAX_VALVE_TIME :	TIME;
		LEVEL_DELAY_TIME :	TIME;
		VALVE :	BOOL;
		ALARM :	BOOL;
		STATUS :	BYTE;

		func_block : TANK_LEVEL_Block;
	END_VAR
	func_block.LEVEL := LEVEL;
	func_block.LEAK := LEAK;
	func_block.ACLR := ACLR ;
	func_block.MAX_VALVE_TIME := MAX_VALVE_TIME;
	func_block.LEVEL_DELAY_TIME := LEVEL_DELAY_TIME ;
	func_block();
	VALVE  := func_block.VALVE;
	ALARM  := func_block.ALARM;
	STATUS  := func_block.STATUS;
END_PROGRAM

CONFIGURATION Config0
	VAR_GLOBAL
		PLC_TICKS_PER_SEC :	INT;
		PLC_SYS_TICK_CNT :	DINT;
	END_VAR
  	RESOURCE Res0 ON PLC
    	TASK task0(INTERVAL := T#20ms,PRIORITY := 0);
    	PROGRAM instance0 WITH task0 : program0;
  	END_RESOURCE
END_CONFIGURATION

(* ---- TC_MS.ST ---- *)
FUNCTION_BLOCK T_PLC_MS_block

	VAR_OUTPUT
		T_PLC_MS :	UDINT;
	END_VAR

	VAR_EXTERNAL
		PLC_TICKS_PER_SEC :	INT;
		PLC_SYS_TICK_CNT :	DINT;
	END_VAR

	VAR
		debug :	BOOL;(*Debug-Mode ON / OFF*)
		N :	INT;(*Debug-Faktor*)
		Offset :	UDINT;(*Debug-Offset*)
		temp :	DWORD := DWORD#1;(*Debug-Offset*)
		mode :	BOOL;(*modus*)
		faktor :	UDINT;(*Systemtakt-Faktor*)
		init :	BOOL;
		v_plc_ticks_per_sec :	UDINT;
		base :	UDINT := UDINT#1000;
	END_VAR

	IF init = FALSE THEN
		v_plc_ticks_per_sec := INT_TO_UDINT(PLC_TICKS_PER_SEC);
		IF v_plc_ticks_per_sec = UDINT#1024 THEN
			faktor := UDINT#1;
			mode := FALSE;
		ELSIF v_plc_ticks_per_sec > UDINT#0 THEN
			IF v_plc_ticks_per_sec <= base THEN
				faktor := base / v_plc_ticks_per_sec;
				mode := FALSE;
			ELSE
				faktor := v_plc_ticks_per_sec / base;
				mode := TRUE;
			END_IF;
		ELSE
			faktor := UDINT#1;
		END_IF;
		init := TRUE;
	END_IF;

	IF mode THEN
		T_PLC_MS := DINT_TO_UDINT(PLC_SYS_TICK_CNT) / faktor;
	ELSE
		T_PLC_MS := DINT_TO_UDINT(PLC_SYS_TICK_CNT) * faktor;
	END_IF;

	IF debug THEN
		T_PLC_MS := (DWORD_TO_UDINT(SHL(UDINT_TO_DWORD(T_PLC_MS),N) OR SHL(temp,N)) - UDINT#1) + Offset;
	END_IF;

END_FUNCTION_BLOCK

FUNCTION_BLOCK TC_MS_Block

	VAR_OUTPUT
		TC :	DWORD;
	END_VAR

	VAR
		init :	BOOL;
		tx :	UDINT;
		last :	UDINT;
		T_PLC_MS :	T_PLC_MS_block;
	END_VAR

	T_PLC_MS();
	tx:= T_PLC_MS.T_PLC_MS;

	IF NOT init THEN
		init := TRUE;
		TC := DWORD#0;
	ELSE
		tc := UDINT_TO_DWORD(tx - last);
	END_IF;
	last := tx;

END_FUNCTION_BLOCK

PROGRAM program0

	VAR
		TC :	DWORD;
		func_block : TC_MS_Block;
	END_VAR
		func_block();
		TC := func_block.TC;

END_PROGRAM

CONFIGURATION Config0

	VAR_GLOBAL
		PLC_TICKS_PER_SEC :	INT;
		PLC_SYS_TICK_CNT :	DINT;
	END_VAR

  	RESOURCE Res0 ON PLC
    	TASK task0(INTERVAL := T#20ms,PRIORITY := 0);
    	PROGRAM instance0 WITH task0 : program0;
  	END_RESOURCE

END_CONFIGURATION

(* ---- TC_S.ST ---- *)
FUNCTION_BLOCK T_PLC_US_Block
	VAR_OUTPUT
		T_PLC_US :	UDINT;
	END_VAR

	VAR_EXTERNAL
		PLC_TICKS_PER_SEC :	INT;
		PLC_SYS_TICK_CNT :	DINT;
	END_VAR

	VAR
		debug :	BOOL;
		N :	INT;
		Offset :	UDINT;
		temp :	DWORD := DWORD#1;
		mode :	BOOL;
		faktor :	UDINT;
		init :	BOOL;
		v_plc_ticks_per_sec :	UDINT;
		base :	UDINT := UDINT#1000000;
	END_VAR

	IF init = FALSE THEN
		v_plc_ticks_per_sec := INT_TO_UDINT(PLC_TICKS_PER_SEC);
		IF v_plc_ticks_per_sec = UDINT#1024 THEN
			faktor := UDINT#1000;
			mode := FALSE;
		ELSIF v_plc_ticks_per_sec > UDINT#0 THEN
			IF v_plc_ticks_per_sec <= base THEN
				faktor := base / v_plc_ticks_per_sec;
				mode := FALSE;
			ELSE
				faktor := v_plc_ticks_per_sec / base;
				mode := TRUE;
			END_IF;
		ELSE
			faktor := UDINT#1;
		END_IF;
		init := TRUE;
	END_IF;

	IF mode THEN
		T_PLC_US := DINT_TO_UDINT(PLC_SYS_TICK_CNT) / faktor;
	ELSE
		T_PLC_US := DINT_TO_UDINT(PLC_SYS_TICK_CNT) * faktor;
	END_IF;

	IF debug THEN
		T_PLC_US := (DWORD_TO_UDINT(SHL(UDINT_TO_DWORD(T_PLC_US),N) OR SHL(temp,N)) - UDINT#1) + Offset;
	END_IF;
END_FUNCTION_BLOCK

FUNCTION_BLOCK TC_S_Block

	VAR_OUTPUT
		TC :	REAL;
	END_VAR

	VAR
		init :	BOOL;
		tx :	UDINT;
		last :	UDINT;
		T_PLC_US :	T_PLC_US_Block;
	END_VAR

	T_PLC_US();
	tx:= T_PLC_US.T_PLC_US;

	IF NOT init THEN
		init := TRUE;
		TC := 0.0;
	ELSE
		tc := UDINT_TO_REAL(tx - last) * 1.0E-6;
	END_IF;
	last := tx;

END_FUNCTION_BLOCK

PROGRAM program0

	VAR
		TC :	REAL;
		func_block : TC_S_Block;
	END_VAR
		func_block();
		TC := func_block.TC;

END_PROGRAM

CONFIGURATION Config0

	VAR_GLOBAL
		PLC_TICKS_PER_SEC :	INT;
		PLC_SYS_TICK_CNT :	DINT;
	END_VAR

	RESOURCE Res0 ON PLC
		TASK task0(INTERVAL := T#20ms,PRIORITY := 0);
		PROGRAM instance0 WITH task0 : program0;
	END_RESOURCE

END_CONFIGURATION

(* ---- TC_US.ST ---- *)
FUNCTION_BLOCK T_PLC_US_Block
	VAR_OUTPUT
		T_PLC_US :	UDINT;
	END_VAR

	VAR_EXTERNAL
		PLC_TICKS_PER_SEC :	INT;
		PLC_SYS_TICK_CNT :	DINT;
	END_VAR

	VAR
		debug :	BOOL;
		N :	INT;
		Offset :	UDINT;
		temp :	DWORD := DWORD#1;
		mode :	BOOL;
		faktor :	UDINT;
		init :	BOOL;
		v_plc_ticks_per_sec :	UDINT;
		base :	UDINT := UDINT#1000000;
	END_VAR

	IF init = FALSE THEN
		v_plc_ticks_per_sec := INT_TO_UDINT(PLC_TICKS_PER_SEC);
		IF v_plc_ticks_per_sec = UDINT#1024 THEN
			faktor := UDINT#1000;
			mode := FALSE;
		ELSIF v_plc_ticks_per_sec > UDINT#0 THEN
			IF v_plc_ticks_per_sec <= base THEN
				faktor := base / v_plc_ticks_per_sec;
				mode := FALSE;
			ELSE
				faktor := v_plc_ticks_per_sec / base;
				mode := TRUE;
			END_IF;
		ELSE
			faktor := UDINT#1;
		END_IF;
		init := TRUE;
	END_IF;

	IF mode THEN
		T_PLC_US := DINT_TO_UDINT(PLC_SYS_TICK_CNT) / faktor;
	ELSE
		T_PLC_US := DINT_TO_UDINT(PLC_SYS_TICK_CNT) * faktor;
	END_IF;

	IF debug THEN
		T_PLC_US := (DWORD_TO_UDINT(SHL(UDINT_TO_DWORD(T_PLC_US),N) OR SHL(temp,N)) - UDINT#1) + Offset;
	END_IF;
END_FUNCTION_BLOCK

FUNCTION_BLOCK TC_US_Block
	VAR_OUTPUT
		TC :	DWORD;
	END_VAR

	VAR
		init :	BOOL;
		tx :	UDINT;
		last :	UDINT;
		T_PLC_US :	T_PLC_US_Block;
	END_VAR

	T_PLC_US();
	tx:= T_PLC_US.T_PLC_US;

	IF NOT init THEN
		init := TRUE;
		TC := DWORD#0;
	ELSE
		tc := UDINT_TO_DWORD(tx - last);
	END_IF;
	last := tx;
END_FUNCTION_BLOCK

PROGRAM program0

	VAR
		TC : DWORD;
		func_block : TC_US_Block;
	END_VAR
		func_block();
		TC := func_block.TC;

END_PROGRAM

CONFIGURATION Config0
	VAR_GLOBAL
		PLC_TICKS_PER_SEC :	INT;
		PLC_SYS_TICK_CNT :	DINT;
	END_VAR

	RESOURCE Res0 ON PLC
		TASK task0(INTERVAL := T#20ms,PRIORITY := 0);
		PROGRAM instance0 WITH task0 : program0;
	END_RESOURCE
END_CONFIGURATION

(* ---- TEMP_EXT.ST ---- *)
FUNCTION UDINT_TO_TIME2:TIME

	VAR_INPUT
		IN :	UDINT;
	END_VAR

	UDINT_TO_TIME2 := DINT_TO_TIME(UDINT_TO_DINT(IN));

END_FUNCTION

FUNCTION_BLOCK T_PLC_MS_block
	VAR_OUTPUT
		T_PLC_MS :	UDINT;
	END_VAR

	VAR_EXTERNAL
		PLC_TICKS_PER_SEC :	INT;
		PLC_SYS_TICK_CNT :	DINT;
	END_VAR

	VAR
		debug :	BOOL;(*Debug-Mode ON / OFF*)
		N :	INT;(*Debug-Faktor*)
		Offset :	UDINT;(*Debug-Offset*)
		temp :	DWORD := DWORD#1;(*Debug-Offset*)
		mode :	BOOL;(*modus*)
		faktor :	UDINT;(*Systemtakt-Faktor*)
		init :	BOOL;
		v_plc_ticks_per_sec :	UDINT;
		base :	UDINT := UDINT#1000;
	END_VAR

	IF init = FALSE THEN
		v_plc_ticks_per_sec := INT_TO_UDINT(PLC_TICKS_PER_SEC);
		IF v_plc_ticks_per_sec = UDINT#1024 THEN
			faktor := UDINT#1;
			mode := FALSE;
		ELSIF v_plc_ticks_per_sec > UDINT#0 THEN
			IF v_plc_ticks_per_sec <= base THEN
				faktor := base / v_plc_ticks_per_sec;
				mode := FALSE;
			ELSE
				faktor := v_plc_ticks_per_sec / base;
				mode := TRUE;
			END_IF;
		ELSE
			faktor := UDINT#1;
		END_IF;
		init := TRUE;
	END_IF;

	IF mode THEN
		T_PLC_MS := DINT_TO_UDINT(PLC_SYS_TICK_CNT) / faktor;
	ELSE
		T_PLC_MS := DINT_TO_UDINT(PLC_SYS_TICK_CNT) * faktor;
	END_IF;

	IF debug THEN
		T_PLC_MS := (DWORD_TO_UDINT(SHL(UDINT_TO_DWORD(T_PLC_MS),N) OR SHL(temp,N)) - UDINT#1) + Offset;
	END_IF;
END_FUNCTION_BLOCK

FUNCTION _INT_TO_UDINT:UDINT
	VAR_INPUT
		IN :	INT;
	END_VAR

	_INT_TO_UDINT := DINT_TO_UDINT(INT_TO_DINT(IN));
END_FUNCTION

FUNCTION SET_DATE:UDINT

	VAR_INPUT
		YEAR :	INT;
		MONTH :	INT;
		DAY :	INT;
	END_VAR

	VAR
		count :	INT;
	END_VAR

	IF month > 2 THEN
		count := (month - 1) * 30;
		IF month > 7 THEN
			count := count + DWORD_TO_INT(SHR(DINT_TO_DWORD(INT_TO_DINT(month) - INT_TO_DINT(3)),1));
		ELSE
			count := count + DWORD_TO_INT(SHR(DINT_TO_DWORD(INT_TO_DINT(month) - INT_TO_DINT(4)),1));
		END_IF;
		IF SHL(INT_TO_WORD(year),14) = WORD#0 THEN
			count := count + 1;
		END_IF;
	ELSE
		count := (month - 1) * 31;
	END_IF;
	SET_DATE := (_INT_TO_UDINT(count + day - 1) + DWORD_TO_UDINT(SHR(UDINT_TO_DWORD(_INT_TO_UDINT(year) * UDINT#1461 - UDINT#2878169), 2))) * UDINT#86400;

END_FUNCTION

FUNCTION LEAP_OF_DATE:BOOL

	VAR_INPUT
		IDATE :	UDINT;
	END_VAR

	LEAP_OF_DATE := SHL(UDINT_TO_DWORD((idate + UDINT#43200) / UDINT#31557600), 30) = DWORD#16#80000000;

END_FUNCTION

FUNCTION DAY_OF_YEAR:INT
	VAR_INPUT
		IDATE :	DATE;
	END_VAR

	DAY_OF_YEAR := UDINT_TO_INT((DATE_TO_UDINT(idate) / UDINT#86400) MOD UDINT#1461);
	IF DAY_OF_YEAR > 729 THEN
		IF DAY_OF_YEAR > 1095 THEN DAY_OF_YEAR := DAY_OF_YEAR - 1095; ELSE DAY_OF_YEAR := DAY_OF_YEAR - 729; END_IF;
	ELSIF DAY_OF_YEAR > 364 THEN
		DAY_OF_YEAR := DAY_OF_YEAR - 364;
	ELSE
		DAY_OF_YEAR := DAY_OF_YEAR + 1;
	END_IF;
END_FUNCTION

FUNCTION DAY_OF_YEAR_UDINT:INT
	VAR_INPUT
		IDATE :	UDINT;
	END_VAR

	DAY_OF_YEAR_UDINT := UDINT_TO_INT((idate / UDINT#86400) MOD UDINT#1461);
	IF DAY_OF_YEAR_UDINT > 729 THEN
		IF DAY_OF_YEAR_UDINT > 1095 THEN DAY_OF_YEAR_UDINT := DAY_OF_YEAR_UDINT - 1095; ELSE DAY_OF_YEAR_UDINT := DAY_OF_YEAR_UDINT - 729; END_IF;
	ELSIF DAY_OF_YEAR_UDINT > 364 THEN
		DAY_OF_YEAR_UDINT := DAY_OF_YEAR_UDINT - 364;
	ELSE
		DAY_OF_YEAR_UDINT := DAY_OF_YEAR_UDINT + 1;
	END_IF;
END_FUNCTION

FUNCTION MONTH_OF_DATE_UDINT:INT

	VAR_INPUT
		IDATE :	UDINT;
	END_VAR

	MONTH_OF_DATE_UDINT := DAY_OF_YEAR_UDINT(idate);
	IF MONTH_OF_DATE_UDINT < 32 THEN
		MONTH_OF_DATE_UDINT := 1;
	ELSIF LEAP_OF_DATE(IDATE) THEN
		MONTH_OF_DATE_UDINT := (MONTH_OF_DATE_UDINT * 53 + 1668) / 1623;
	ELSE
		MONTH_OF_DATE_UDINT := (MONTH_OF_DATE_UDINT * 53 + 1700) / 1620;
	END_IF;

END_FUNCTION

FUNCTION DAY_OF_MONTH:INT
	VAR_INPUT
		IDATE :	UDINT;
	END_VAR

	day_of_month := day_of_year_UDINT(idate);

	IF leap_of_Date(idate) THEN
		CASE day_of_month OF
			32..60	:	day_of_month := day_of_month - 31;
			61..91	:	day_of_month := day_of_month - 60;
			92..121 :	day_of_month := day_of_month - 91;
			122..152:	day_of_month := day_of_month - 121;
			153..182:	day_of_month := day_of_month - 152;
			183..213:	day_of_month := day_of_month - 182;
			214..244:	day_of_month := day_of_month - 213;
			245..274:	day_of_month := day_of_month - 244;
			275..305:	day_of_month := day_of_month - 274;
			306..335:	day_of_month := day_of_month - 305;
			336..366:	day_of_month := day_of_month - 335;
		END_CASE;
	ELSE
		CASE day_of_month OF
			32..59	:	day_of_month := day_of_month - 31;
			60..90	:	day_of_month := day_of_month - 59;
			91..120 :	day_of_month := day_of_month - 90;
			121..151:	day_of_month := day_of_month - 120;
			152..181:	day_of_month := day_of_month - 151;
			182..212:	day_of_month := day_of_month - 181;
			213..243:	day_of_month := day_of_month - 212;
			244..273:	day_of_month := day_of_month - 243;
			274..304:	day_of_month := day_of_month - 273;
			305..334:	day_of_month := day_of_month - 304;
			335..365:	day_of_month := day_of_month - 334;
		END_CASE;
	END_IF;

END_FUNCTION

FUNCTION MID3:REAL

	VAR_INPUT
		IN1 :	REAL;
		IN2 :	REAL;
		IN3 :	REAL;
	END_VAR

	VAR
		_IN1 :	REAL;
		_IN2 :	REAL;
		_IN3 :	REAL;
	END_VAR

	_IN1 := IN1;
	_IN2 := IN2;
	_IN3 := IN3;

	IF _IN1 > _IN2 THEN MID3 := _IN1; _IN1 := _IN2; _IN2 := MID3; END_IF;
	IF _IN2 > _IN3 THEN _IN2 := _IN3; END_IF;
	MID3 := SEL(_IN1 > _IN2, _IN2, _IN1);

END_FUNCTION

FUNCTION _BYTE_TO_INT:INT
	VAR_INPUT
		IN :	BYTE;
	END_VAR

	_BYTE_TO_INT := USINT_TO_INT(BYTE_TO_USINT(IN));
END_FUNCTION

FUNCTION MULTI_IN:REAL

	VAR_INPUT
		IN_1 :	REAL;
		IN_2 :	REAL;
		IN_3 :	REAL;
		DEFAULT :	REAL;
		IN_MIN :	REAL;
		IN_MAX :	REAL;
		MODE :	BYTE;
	END_VAR

	VAR
		count :	INT;
		F1 :	BOOL;
		F2 :	BOOL;
		F3 :	BOOL;
	END_VAR

	F1 :=  in_1 > in_min AND in_1 < in_max;
	F2 :=  in_2 > in_min AND in_2 < in_max;
	F3 :=  in_3 > in_min AND in_3 < in_max;

	CASE _BYTE_TO_INT(mode) OF
	0:	count := 0;
		IF F1 THEN
			count := count + 1;
			MULTI_IN := in_1;
		ELSE
			MULTI_IN := 0.0;
		END_IF;
		IF F2 THEN
			count := count + 1;
			MULTI_IN := MULTI_IN + in_2;
		END_IF;
		IF F3 THEN
			count := count + 1;
			MULTI_IN := MULTI_IN + in_3;
		END_IF;
		MULTI_IN := SEL_REAL(count = 0, MULTI_IN / INT_TO_REAL(count), default);

	1:	MULTI_IN := SEL_REAL(F1, default, IN_1);

	2:	MULTI_IN := SEL_REAL(F2, default, IN_2);

	3:	MULTI_IN := SEL_REAL(F3, default, IN_3);

	4:	MULTI_IN := default;

	5:	MULTI_IN := SEL_REAL(F1, in_max, IN_1);
		IF F2 AND in_2 < MULTI_IN THEN MULTI_IN := in_2; END_IF;
		IF F3 AND in_3 < MULTI_IN THEN MULTI_IN := in_3; END_IF;
		IF MULTI_IN = in_max THEN MULTI_IN := default; END_IF;

	6:	MULTI_IN := SEL_REAL(F1, in_min, IN_1);
		IF F2 AND in_2 > MULTI_IN THEN MULTI_IN := in_2; END_IF;
		IF F3 AND in_3 > MULTI_IN THEN MULTI_IN := in_3; END_IF;
		IF MULTI_IN = in_min THEN MULTI_IN := default; END_IF;

	7:	IF F1 AND F2 AND F3 THEN MULTI_IN := MID3(in_1, in_2, in_3);
		ELSIF F1 AND F2 THEN MULTI_IN := MIN(in_1, in_2);
		ELSIF F1 AND F3 THEN MULTI_IN := MIN(in_1, in_3);
		ELSIF F2 AND F3 THEN MULTI_IN := MIN(in_2, in_3);
		ELSIF F1 THEN MULTI_IN := in_1;
		ELSIF F2 THEN MULTI_IN := in_2;
		ELSIF F3 THEN MULTI_IN := in_3;
		ELSE MULTI_IN := default;
		END_IF;

	END_CASE;

END_FUNCTION

FUNCTION _DT_TO_DATE_B:UDINT

	VAR_INPUT
		_INN :	UDINT;
	END_VAR

	_DT_TO_DATE_B := (_INN / UDINT#86400) * UDINT#86400;
END_FUNCTION

FUNCTION DT_TO_TOD2:UDINT
	VAR_INPUT
		IN :	UDINT;
	END_VAR

	DT_TO_TOD2 := (IN MOD UDINT#86400) * UDINT#1000;
END_FUNCTION

FUNCTION_BLOCK TEMP_EXT_Block

	VAR_INPUT
		T_EXT1 :	REAL;
		T_EXT2 :	REAL;
		T_EXT3 :	REAL;
		T_EXT_CONFIG :	BYTE := 0;
		DT_IN :	UDINT;
		T_EXT_MIN :	REAL := REAL#-40.0;
		T_EXT_MAX :	REAL := REAL#60.0;
		T_EXT_DEFAULT :	REAL := REAL#-10.0;
		HEAT_PERIOD_START :	UDINT := UDINT#20995200;
		HEAT_PERIOD_STOP :	UDINT := UDINT#10281600;
		COOL_PERIOD_START :	UDINT := UDINT#07776000;
		COOL_PERIOD_STOP :	UDINT := UDINT#23500800;
		HEAT_START_TEMP_DAY :	REAL := REAL#15.0;
		HEAT_START_TEMP_NIGHT :	REAL := REAL#10.0;
		HEAT_STOP_TEMP :	REAL := REAL#18.0;
		COOL_START_TEMP_DAY :	REAL := REAL#26.0;
		COOL_START_TEMP_NIGHT :	REAL := REAL#26.0;
		COOL_STOP_TEMP :	REAL := REAL#24.0;
		START_DAY :	UDINT := UDINT#32400000;
		START_NIGHT :	UDINT := UDINT#75600000;
		CYCLE_TIME :	TIME := t#10m;
	END_VAR

	VAR_OUTPUT
		T_EXT :	REAL;
		HEAT :	BOOL;
		COOL :	BOOL;
	END_VAR

	VAR
		tx :	TIME;
		last_run :	TIME;
		init :	BOOL;
		cool_start :	UDINT;
		cool_stop :	UDINT;
		heat_start :	UDINT;
		heat_stop :	UDINT;
		xdate :	UDINT;
		day :	BOOL;
		T_PLC_MS :	T_PLC_MS_Block;
	END_VAR

	IF NOT init THEN
		init := TRUE;
		heat_start := SET_DATE(1972,MONTH_OF_DATE_UDINT(heat_period_start),DAY_OF_MONTH(heat_period_start));
		heat_stop := SET_DATE(1972,MONTH_OF_DATE_UDINT(heat_period_stop),DAY_OF_MONTH(heat_period_stop));
		cool_start := SET_DATE(1972,MONTH_OF_DATE_UDINT(cool_period_start),DAY_OF_MONTH(cool_period_start));
		cool_stop := SET_DATE(1972,MONTH_OF_DATE_UDINT(cool_period_stop),DAY_OF_MONTH(cool_period_stop));
	END_IF;

	T_PLC_MS();
	tx:= UDINT_TO_TIME(T_PLC_MS.T_PLC_MS);

	IF tx - last_run < cycle_time THEN RETURN; END_IF;

	xdate := SET_DATE(1972,MONTH_OF_DATE_UDINT(_DT_TO_DATE_B(dt_in)),DAY_OF_MONTH(_DT_TO_DATE_B(dt_in)));
	day := DT_TO_TOD2(dt_in) >= start_day AND  DT_TO_TOD2(dt_in) < start_night;

	t_ext := MULTI_IN(t_ext1, t_ext2, t_ext3, t_ext_default, t_ext_min, t_ext_max, t_ext_config);

	IF (heat_start <= heat_stop AND xdate >= heat_start AND xdate <= heat_stop) OR (heat_start > heat_stop AND (xdate >= heat_start OR xdate <= heat_stop)) THEN
		IF day AND t_ext <= heat_start_temp_day THEN
			heat := TRUE;
		ELSIF NOT day AND t_ext <= heat_start_temp_night THEN
			heat := TRUE;
		ELSIF t_ext >= heat_stop_temp THEN
			heat := FALSE;
		END_IF;
	ELSE
		heat := FALSE;
	END_IF;

	IF (cool_start <= cool_stop AND xdate >= cool_start AND xdate <= cool_stop) OR (cool_start > cool_stop AND (xdate >= cool_start OR xdate <= cool_stop)) THEN
		IF day AND t_ext >= cool_start_temp_day THEN
			cool := TRUE;
		ELSIF NOT day AND t_ext >= cool_start_temp_night THEN
			cool := TRUE;
		ELSIF t_ext <= cool_stop_temp THEN
			cool := FALSE;
		END_IF;
	ELSE
		cool := FALSE;
	END_IF;

	last_run := tx;

END_FUNCTION_BLOCK

PROGRAM program0
	VAR
		T_EXT1 :	REAL;
		T_EXT2 :	REAL;
		T_EXT3 :	REAL;
		T_EXT_CONFIG :	BYTE := 0;
		DT_IN :	UDINT;
		T_EXT_MIN :	REAL := REAL#-40.0;
		T_EXT_MAX :	REAL := REAL#60.0;
		T_EXT_DEFAULT :	REAL := REAL#-10.0;
		HEAT_PERIOD_START :	UDINT := UDINT#20995200;
		HEAT_PERIOD_STOP :	UDINT := UDINT#10281600;
		COOL_PERIOD_START :	UDINT := UDINT#07776000;
		COOL_PERIOD_STOP :	UDINT := UDINT#23500800;
		HEAT_START_TEMP_DAY :	REAL := REAL#15.0;
		HEAT_START_TEMP_NIGHT :	REAL := REAL#10.0;
		HEAT_STOP_TEMP :	REAL := REAL#18.0;
		COOL_START_TEMP_DAY :	REAL := REAL#26.0;
		COOL_START_TEMP_NIGHT :	REAL := REAL#26.0;
		COOL_STOP_TEMP :	REAL := REAL#24.0;
		START_DAY :	UDINT := UDINT#32400000;
		START_NIGHT :	UDINT := UDINT#75600000;
		CYCLE_TIME :	TIME := t#10m;
		T_EXT :	REAL;
		HEAT :	BOOL;
		COOL :	BOOL;

		func_block : TEMP_EXT_Block;
	END_VAR

	func_block.T_EXT1 := T_EXT1;
	func_block.T_EXT2 := T_EXT2;
	func_block.T_EXT3 := T_EXT3 ;
	func_block.T_EXT_CONFIG := T_EXT_CONFIG;
	func_block.DT_IN := DT_IN;
	func_block.T_EXT_MIN := T_EXT_MIN ;
	func_block.T_EXT_MAX := T_EXT_MAX;
	func_block.T_EXT_DEFAULT := T_EXT_DEFAULT;
	func_block.HEAT_PERIOD_START := HEAT_PERIOD_START ;
	func_block.HEAT_PERIOD_STOP := HEAT_PERIOD_STOP;
	func_block.COOL_PERIOD_START := COOL_PERIOD_START;
	func_block.COOL_PERIOD_STOP := COOL_PERIOD_STOP ;
	func_block.HEAT_START_TEMP_DAY := HEAT_START_TEMP_DAY;
	func_block.HEAT_START_TEMP_NIGHT := HEAT_START_TEMP_NIGHT;
	func_block.HEAT_STOP_TEMP := HEAT_STOP_TEMP ;
	func_block.COOL_START_TEMP_DAY := COOL_START_TEMP_DAY;
	func_block.COOL_START_TEMP_NIGHT := COOL_START_TEMP_NIGHT;
	func_block.COOL_STOP_TEMP:= COOL_STOP_TEMP ;
	func_block.START_DAY := START_DAY;
	func_block.START_NIGHT := START_NIGHT;
	func_block.CYCLE_TIME:= CYCLE_TIME ;

	func_block();
	T_EXT  := func_block.T_EXT;
	HEAT  := func_block.HEAT;
	COOL  := func_block.COOL;

END_PROGRAM

CONFIGURATION Config0
	VAR_GLOBAL
		PLC_TICKS_PER_SEC :	INT;
		PLC_SYS_TICK_CNT :	DINT;
	END_VAR
  	RESOURCE Res0 ON PLC
    	TASK task0(INTERVAL := T#20ms,PRIORITY := 0);
    	PROGRAM instance0 WITH task0 : program0;
  	END_RESOURCE
END_CONFIGURATION

(* ---- TEMPERATURE.ST ---- *)
FUNCTION_BLOCK TEMPERATURE

	VAR_INPUT
		K :	REAL;
		C :	REAL := -273.15;
		F :	REAL := -459.67;
		RE :	REAL := -218.52;
		RA :	REAL := 0.0;
	END_VAR

	VAR_OUTPUT
		YK :	REAL;
		YC :	REAL;
		YF :	REAL;
		YRE :	REAL;
		YRA :	REAL;
	END_VAR

	YK := K + (C + 273.15) + (F + 459.67) * 0.555555555555 + (Re * 1.25 + 273.15) + (Ra * 0.555555555555);
	YC := YK -273.15;
	YF := YK * 1.8 - 459.67;
	YRe := (YK - 273.15) * 0.8;
	YRa := YK * 1.8;

END_FUNCTION_BLOCK

PROGRAM program0
  VAR
	K :	REAL;
	C :	REAL := -273.15;
	F :	REAL := -459.67;
	RE :	REAL := -218.52;
	RA :	REAL := 0.0;
	YK :	REAL;
	YC :	REAL;
	YF :	REAL;
	YRE :	REAL;
	YRA :	REAL;
	func_block : TEMPERATURE;
  END_VAR
	func_block.K  :=K;
	func_block.C  :=C;
	func_block.F  :=F;
	func_block.RE  :=RE;
	func_block.RA  :=RA;
	func_block();
	YK := func_block.YK;
	YC := func_block.YC;
	YF := func_block.YF;
	YRE := func_block.YRE;
	YRA := func_block.YRA;

END_PROGRAM

CONFIGURATION Config0
	RESOURCE Res0 ON PLC
		TASK task0(INTERVAL := T#20ms,PRIORITY := 0);
		PROGRAM instance0 WITH task0 : program0;
	END_RESOURCE
END_CONFIGURATION

(* ---- TICKER.ST ---- *)
TYPE
	oscat_delay_buf             : ARRAY [0..31]   OF REAL;
END_TYPE

FUNCTION INC1:INT

	VAR_INPUT
		X :	INT;
		N :	INT;
	END_VAR

	IF X >= N - 1 THEN
		INC1 := 0;
	ELSE
		INC1 := X + 1;
	END_IF;
END_FUNCTION

FUNCTION_BLOCK DELAY

	VAR_INPUT
		IN :	REAL;
		N :	INT;
		RST :	BOOL;
	END_VAR

	VAR_OUTPUT
		OUT :	REAL;
	END_VAR

	VAR
		buf :	oscat_delay_buf;
		i :	INT;
		init :	BOOL;
		stop :	INT;
	END_VAR

	stop := LIMIT(0,N,32) - 1;
	IF rst OR NOT init THEN
		init := TRUE;
		FOR i := 0 TO stop DO buf[i] := in; END_FOR;
		out := in;
		i := 0;
	ELSIF stop < 0 THEN
		out := in;
	ELSE
		out := buf[i];
		buf[i] := in;
		i := INC1(i, N);
	END_IF;

END_FUNCTION_BLOCK

FUNCTION_BLOCK TICKER

	VAR_INPUT
		N :	INT;
		PT :	TIME;
		TEXT :	STRING;
	END_VAR

	VAR_OUTPUT
		DISPLAY :	STRING;
	END_VAR

	VAR
		_delay :	TP;
		rollout :	STRING;
		text_len :	INT;
		rollout_step :	INT;
		_step :	INT;
	END_VAR

	text_len := LEN(text);

	IF N < text_len THEN
		IF NOT _delay.Q THEN

			IF _step > text_len THEN
				rollout_step := 0;
				rollout := '';
				_step := 0;
			END_IF;

			IF _step + N > text_len THEN
				_step := _step + 1;
				rollout_step := rollout_step +1;
				display := MID(text, N - rollout_step, _step);
				rollout := CONCAT(rollout,'#');
				display := CONCAT(display,rollout);
			ELSE
				_step := _step + 1;
				display := MID(text, N, _step);
			END_IF;
			_delay(TRUE, PT);
		ELSE
			_delay(FALSE);
		END_IF;
	ELSE
		display := text;
	END_IF;

END_FUNCTION_BLOCK

PROGRAM program0
	VAR
		N :	INT;
		PT :	TIME;
		TEXT :	STRING;
		DISPLAY :	STRING;
		func_block : TICKER;
  	END_VAR
	func_block.N  :=N;
	func_block.PT  :=PT;
	func_block.TEXT  :=TEXT;
	func_block();
	DISPLAY := func_block.DISPLAY;
END_PROGRAM

CONFIGURATION Config0
	RESOURCE Res0 ON PLC
		TASK task0(INTERVAL := T#20ms,PRIORITY := 0);
		PROGRAM instance0 WITH task0 : program0;
	END_RESOURCE
END_CONFIGURATION

(* ---- TIMER_1.ST ---- *)
FUNCTION TIMECHECK:BOOL

	VAR_INPUT
		TD :	UDINT;
		START :	UDINT;
		STOP :	UDINT;
	END_VAR

	IF stop < start THEN
		TIMECHECK := start <= TD OR  TD < stop;
	ELSE
		TIMECHECK := start <= TD AND TD < stop;
	END_IF;

END_FUNCTION

FUNCTION TIME_TO_TOD:UDINT

	VAR_INPUT
		IN :	TIME;
	END_VAR

	TIME_TO_TOD := DWORD_TO_UDINT(TIME_TO_DWORD(IN));
END_FUNCTION

FUNCTION TOD_TO_TIME:TIME
	VAR_INPUT
		IN :	UDINT;
	END_VAR

	TOD_TO_TIME := DWORD_TO_TIME(UDINT_TO_DWORD(IN));
END_FUNCTION

FUNCTION DAY_OF_WEEK:INT
  VAR_INPUT
    IDATE :	UDINT;
  END_VAR

  DAY_OF_WEEK := UDINT_TO_INT((idate / UDINT#86400 + UDINT#3) MOD UDINT#7) + INT#01;
END_FUNCTION

FUNCTION _DT_TO_DATE_B:UDINT

	VAR_INPUT
		_INN :	UDINT;
	END_VAR

	_DT_TO_DATE_B := (_INN / UDINT#86400) * UDINT#86400;
END_FUNCTION

FUNCTION DT_TO_TOD2:UDINT
	VAR_INPUT
		IN :	UDINT;
	END_VAR

	DT_TO_TOD2 := (IN MOD UDINT#86400) * UDINT#1000;
END_FUNCTION

FUNCTION TIME_TO_TOD2:UDINT

	VAR_INPUT
		IN :	TIME;
	END_VAR

	TIME_TO_TOD2 := DWORD_TO_UDINT(TIME_TO_DWORD(IN));
END_FUNCTION

FUNCTION_BLOCK TIMER_1_Block

	VAR_INPUT
		E :	BOOL := TRUE;
		DTI :	UDINT;
		START :	UDINT;
		DURATION :	TIME;
		DAY :	BYTE := BYTE#2#0111_1111;
	END_VAR

	VAR_OUTPUT
		Q :	BOOL;
		STOP :	TIME;
	END_VAR

	IF E THEN
		stop := TOD_TO_TIME(START) + DURATION;
		IF stop > T#24h THEN stop := stop - T#24h; END_IF;
		Q := TIMECHECK(DT_TO_TOD2(DTI), START, TIME_TO_TOD2(stop)) AND (SHR(BYTE#128, DAY_OF_WEEK(_DT_TO_DATE_B(DTI))) AND DAY) > BYTE#0;
	ELSE
		Q := FALSE;
	END_IF;

END_FUNCTION_BLOCK

PROGRAM program0
	VAR
		E :	BOOL := TRUE;
		DTI :	UDINT;
		START :	UDINT;
		DURATION :	TIME;
		DAY :	BYTE := BYTE#2#0111_1111;
		Q :	BOOL;
		STOP :	TIME;

		func_block : TIMER_1_Block;
	END_VAR
	func_block.E := E;
	func_block.DTI := DTI;
	func_block.START := START ;
	func_block.DURATION    := DURATION    ;
	func_block.DAY := DAY;

	func_block();
	Q  := func_block.Q;
	STOP  := func_block.STOP;
END_PROGRAM

CONFIGURATION Config0
	RESOURCE Res0 ON PLC
		TASK task0(INTERVAL := T#20ms,PRIORITY := 0);
		PROGRAM instance0 WITH task0 : program0;
	END_RESOURCE
END_CONFIGURATION

(* ---- TIMER_2.ST ---- *)
FUNCTION UDINT_TO_TIME2:TIME

	VAR_INPUT
		IN :	UDINT;
	END_VAR

	UDINT_TO_TIME2 := DINT_TO_TIME(UDINT_TO_DINT(IN));

END_FUNCTION

FUNCTION_BLOCK T_PLC_MS_block
	VAR_OUTPUT
		T_PLC_MS :	UDINT;
	END_VAR

	VAR_EXTERNAL
		PLC_TICKS_PER_SEC :	INT;
		PLC_SYS_TICK_CNT :	DINT;
	END_VAR

	VAR
		debug :	BOOL;(*Debug-Mode ON / OFF*)
		N :	INT;(*Debug-Faktor*)
		Offset :	UDINT;(*Debug-Offset*)
		temp :	DWORD := DWORD#1;(*Debug-Offset*)
		mode :	BOOL;(*modus*)
		faktor :	UDINT;(*Systemtakt-Faktor*)
		init :	BOOL;
		v_plc_ticks_per_sec :	UDINT;
		base :	UDINT := UDINT#1000;
	END_VAR

	IF init = FALSE THEN
		v_plc_ticks_per_sec := INT_TO_UDINT(PLC_TICKS_PER_SEC);
		IF v_plc_ticks_per_sec = UDINT#1024 THEN
			faktor := UDINT#1;
			mode := FALSE;
		ELSIF v_plc_ticks_per_sec > UDINT#0 THEN
			IF v_plc_ticks_per_sec <= base THEN
				faktor := base / v_plc_ticks_per_sec;
				mode := FALSE;
			ELSE
				faktor := v_plc_ticks_per_sec / base;
				mode := TRUE;
			END_IF;
		ELSE
			faktor := UDINT#1;
		END_IF;
		init := TRUE;
	END_IF;

	IF mode THEN
		T_PLC_MS := DINT_TO_UDINT(PLC_SYS_TICK_CNT) / faktor;
	ELSE
		T_PLC_MS := DINT_TO_UDINT(PLC_SYS_TICK_CNT) * faktor;
	END_IF;

	IF debug THEN
		T_PLC_MS := (DWORD_TO_UDINT(SHL(UDINT_TO_DWORD(T_PLC_MS),N) OR SHL(temp,N)) - UDINT#1) + Offset;
	END_IF;
END_FUNCTION_BLOCK

FUNCTION DAY_OF_WEEK:INT
  VAR_INPUT
    IDATE :	UDINT;
  END_VAR

  DAY_OF_WEEK := UDINT_TO_INT((idate / UDINT#86400 + UDINT#3) MOD UDINT#7) + INT#01;
END_FUNCTION

FUNCTION _BYTE_TO_INT:INT
	VAR_INPUT
		IN :	BYTE;
	END_VAR

	_BYTE_TO_INT := USINT_TO_INT(BYTE_TO_USINT(IN));
END_FUNCTION

FUNCTION LEAP_OF_DATE:BOOL

	VAR_INPUT
		IDATE :	UDINT;
	END_VAR

	LEAP_OF_DATE := SHL(UDINT_TO_DWORD((idate + UDINT#43200) / UDINT#31557600), 30) = DWORD#16#80000000;

END_FUNCTION

FUNCTION DAY_OF_YEAR:INT
	VAR_INPUT
		IDATE :	DATE;
	END_VAR

	DAY_OF_YEAR := UDINT_TO_INT((DATE_TO_UDINT(idate) / UDINT#86400) MOD UDINT#1461);
	IF DAY_OF_YEAR > 729 THEN
		IF DAY_OF_YEAR > 1095 THEN DAY_OF_YEAR := DAY_OF_YEAR - 1095; ELSE DAY_OF_YEAR := DAY_OF_YEAR - 729; END_IF;
	ELSIF DAY_OF_YEAR > 364 THEN
		DAY_OF_YEAR := DAY_OF_YEAR - 364;
	ELSE
		DAY_OF_YEAR := DAY_OF_YEAR + 1;
	END_IF;
END_FUNCTION

FUNCTION DAY_OF_YEAR_UDINT:INT
	VAR_INPUT
		IDATE :	UDINT;
	END_VAR

	DAY_OF_YEAR_UDINT := UDINT_TO_INT((idate / UDINT#86400) MOD UDINT#1461);
	IF DAY_OF_YEAR_UDINT > 729 THEN
		IF DAY_OF_YEAR_UDINT > 1095 THEN DAY_OF_YEAR_UDINT := DAY_OF_YEAR_UDINT - 1095; ELSE DAY_OF_YEAR_UDINT := DAY_OF_YEAR_UDINT - 729; END_IF;
	ELSIF DAY_OF_YEAR_UDINT > 364 THEN
		DAY_OF_YEAR_UDINT := DAY_OF_YEAR_UDINT - 364;
	ELSE
		DAY_OF_YEAR_UDINT := DAY_OF_YEAR_UDINT + 1;
	END_IF;
END_FUNCTION

FUNCTION MONTH_OF_DATE_UDINT:INT

	VAR_INPUT
		IDATE :	UDINT;
	END_VAR

	MONTH_OF_DATE_UDINT := DAY_OF_YEAR_UDINT(idate);
	IF MONTH_OF_DATE_UDINT < 32 THEN
		MONTH_OF_DATE_UDINT := 1;
	ELSIF LEAP_OF_DATE(IDATE) THEN
		MONTH_OF_DATE_UDINT := (MONTH_OF_DATE_UDINT * 53 + 1668) / 1623;
	ELSE
		MONTH_OF_DATE_UDINT := (MONTH_OF_DATE_UDINT * 53 + 1700) / 1620;
	END_IF;

END_FUNCTION

FUNCTION DAY_OF_MONTH:INT
	VAR_INPUT
		IDATE :	UDINT;
	END_VAR

	day_of_month := day_of_year_UDINT(idate);

	IF leap_of_Date(idate) THEN
		CASE day_of_month OF
			32..60	:	day_of_month := day_of_month - 31;
			61..91	:	day_of_month := day_of_month - 60;
			92..121 :	day_of_month := day_of_month - 91;
			122..152:	day_of_month := day_of_month - 121;
			153..182:	day_of_month := day_of_month - 152;
			183..213:	day_of_month := day_of_month - 182;
			214..244:	day_of_month := day_of_month - 213;
			245..274:	day_of_month := day_of_month - 244;
			275..305:	day_of_month := day_of_month - 274;
			306..335:	day_of_month := day_of_month - 305;
			336..366:	day_of_month := day_of_month - 335;
		END_CASE;
	ELSE
		CASE day_of_month OF
			32..59	:	day_of_month := day_of_month - 31;
			60..90	:	day_of_month := day_of_month - 59;
			91..120 :	day_of_month := day_of_month - 90;
			121..151:	day_of_month := day_of_month - 120;
			152..181:	day_of_month := day_of_month - 151;
			182..212:	day_of_month := day_of_month - 181;
			213..243:	day_of_month := day_of_month - 212;
			244..273:	day_of_month := day_of_month - 243;
			274..304:	day_of_month := day_of_month - 273;
			305..334:	day_of_month := day_of_month - 304;
			335..365:	day_of_month := day_of_month - 334;
		END_CASE;
	END_IF;

END_FUNCTION

FUNCTION MONTH_OF_DATE:INT

	VAR_INPUT
		IDATE :	DATE;
	END_VAR

	MONTH_OF_DATE := DAY_OF_YEAR(idate);
	IF MONTH_OF_DATE < 32 THEN
		MONTH_OF_DATE := 1;
	ELSIF LEAP_OF_DATE(DATE_TO_UDINT(IDATE)) THEN
		MONTH_OF_DATE := (MONTH_OF_DATE * 53 + 1668) / 1623;
	ELSE
		MONTH_OF_DATE := (MONTH_OF_DATE * 53 + 1700) / 1620;
	END_IF;

END_FUNCTION

FUNCTION TIME_TO_UDINT2:UDINT
	VAR_INPUT
		X :	TIME;
	END_VAR

	TIME_TO_UDINT2 := DINT_TO_UDINT(TIME_TO_DINT(X));
END_FUNCTION

FUNCTION DT_TO_TOD2:UDINT
	VAR_INPUT
		IN :	UDINT;
	END_VAR

	DT_TO_TOD2 := (IN MOD UDINT#86400) * UDINT#1000;
END_FUNCTION

FUNCTION _DT_TO_DATE_B:UDINT

	VAR_INPUT
		_INN :	UDINT;
	END_VAR

	_DT_TO_DATE_B := (_INN / UDINT#86400) * UDINT#86400;
END_FUNCTION

FUNCTION_BLOCK TIMER_2_Block

	VAR_INPUT
		DT_IN :	UDINT;
		START :	UDINT;
		DURATION :	TIME;
		MODE :	BYTE;
		HOLIDAY :	BOOL;
	END_VAR

	VAR_OUTPUT
		Q :	BOOL;
	END_VAR

	VAR
		last_check :	TIME := T#0s;
		dat :	UDINT;
		daytime :	UDINT;
		activation :	TIME;
		tx :	TIME;
		enabled :	BOOL;
		wday :	INT;
		init :	BOOL;
	END_VAR

	VAR RETAIN
		run_date :	UDINT;
	END_VAR

	VAR
		T_PLC_MS :	T_PLC_MS_Block;
	END_VAR

	T_PLC_MS();
	tx:= UDINT_TO_TIME(T_PLC_MS.T_PLC_MS);

	IF NOT init THEN
		init := TRUE;
		last_check := tx - t#100ms;
	END_IF;

	IF tx - last_check < T#100ms THEN RETURN; END_IF;

	dat := _DT_TO_DATE_B(dt_in);
	daytime := DT_TO_TOD2(dt_in);
	wday := DAY_OF_WEEK(dat);

	CASE _BYTE_TO_INT(mode) OF
	1..7:
		enabled := wday = _BYTE_TO_INT(mode);
	11:
		enabled := TRUE;
	12..16:
		enabled := (dat / UDINT#86400) MOD (BYTE_TO_UDINT(mode) - UDINT#10) = UDINT#0;
	20:
		enabled := wday <= 5;
	21:
		enabled := wday > 5;
	22:
		enabled := wday <= 5 AND NOT holiday;
	23:
		enabled := wday > 5 OR holiday;
	24:
		enabled := holiday;
	25:
		enabled := DAY_OF_MONTH(dat) = 1;
	26:
		enabled := day_of_month(dat + TIME_TO_UDINT2(t#1d)) = 1;
	27:
		enabled := DAY_OF_MONTH(dat) = 31 AND MONTH_OF_DATE_UDINT(dat) = 12;
	28:
		enabled := DAY_OF_YEAR_UDINT(dat) = 1;
	ELSE
		enabled := FALSE;
	END_CASE;

	IF enabled AND NOT Q AND daytime >= start AND run_date <> dat THEN
		Q := TRUE;
		activation := tx;
		run_date := dat;
	ELSIF Q AND tx - activation >= duration THEN
		Q := FALSE;
	END_IF;
	last_check := Tx;

END_FUNCTION_BLOCK

PROGRAM program0
	VAR
		DT_IN :	UDINT;
		START :	UDINT;
		DURATION :	TIME;
		MODE :	BYTE;
		HOLIDAY :	BOOL;
		Q :	BOOL;

		func_block : TIMER_2_Block;
	END_VAR
	func_block.DT_IN := DT_IN;
	func_block.START := START;
	func_block.DURATION := DURATION ;
	func_block.MODE    := MODE    ;
	func_block.HOLIDAY := HOLIDAY;

	func_block();
	Q  := func_block.Q;
END_PROGRAM

CONFIGURATION Config0
	VAR_GLOBAL
		PLC_TICKS_PER_SEC :	INT;
		PLC_SYS_TICK_CNT :	DINT;
	END_VAR
  	RESOURCE Res0 ON PLC
    	TASK task0(INTERVAL := T#20ms,PRIORITY := 0);
    	PROGRAM instance0 WITH task0 : program0;
  	END_RESOURCE
END_CONFIGURATION

(* ---- TIMER_EXT.ST ---- *)
FUNCTION_BLOCK MANUAL_2_Block

	VAR_INPUT
		_IN :	BOOL;
		ENA :	BOOL;
		_ON :	BOOL;
		OFF :	BOOL;
		MAN :	BOOL;
	END_VAR

	VAR_OUTPUT
		Q :	BOOL;
		STATUS :	BYTE;
	END_VAR

	IF ena THEN
		IF NOT _ON AND NOT OFF THEN
			Q := _IN;
			STATUS := BYTE#100;
		ELSIF _on AND NOT off THEN
			Q := TRUE;
			STATUS := BYTE#101;
		ELSIF NOT _on AND off THEN
			q := FALSE;
			STATUS := BYTE#102;
		ELSE
			Q := MAN;
			STATUS := BYTE#103;
		END_IF;
	ELSE
		Q := FALSE;
		STATUS := BYTE#104;
	END_IF;

END_FUNCTION_BLOCK

FUNCTION_BLOCK DEBOUNCE_Block

	VAR_INPUT
		IN :	BOOL;
		TD :	TIME;
		PM :	BOOL;
	END_VAR

	VAR_OUTPUT
		Q :	BOOL;
	END_VAR

	VAR
		deb :	TOF;
	END_VAR

	IF NOT deb.Q AND IN THEN
		Q := TRUE;
	ELSIF NOT PM THEN
		Q := deb.Q;
	ELSE
		Q := FALSE;
	END_IF;

END_FUNCTION_BLOCK

FUNCTION_BLOCK T_PLC_MS_block

	VAR_OUTPUT
		T_PLC_MS :	UDINT;
	END_VAR

	VAR_EXTERNAL
		PLC_TICKS_PER_SEC :	INT;
		PLC_SYS_TICK_CNT :	DINT;
	END_VAR

	VAR
		debug :	BOOL;(*Debug-Mode ON / OFF*)
		N :	INT;(*Debug-Faktor*)
		Offset :	UDINT;(*Debug-Offset*)
		temp :	DWORD := DWORD#1;(*Debug-Offset*)
		mode :	BOOL;(*modus*)
		faktor :	UDINT;(*Systemtakt-Faktor*)
		init :	BOOL;
		v_plc_ticks_per_sec :	UDINT;
		base :	UDINT := UDINT#1000;
	END_VAR

	IF init = FALSE THEN
		v_plc_ticks_per_sec := INT_TO_UDINT(PLC_TICKS_PER_SEC);
		IF v_plc_ticks_per_sec = UDINT#1024 THEN
			faktor := UDINT#1;
			mode := FALSE;
		ELSIF v_plc_ticks_per_sec > UDINT#0 THEN
			IF v_plc_ticks_per_sec <= base THEN
				faktor := base / v_plc_ticks_per_sec;
				mode := FALSE;
			ELSE
				faktor := v_plc_ticks_per_sec / base;
				mode := TRUE;
			END_IF;
		ELSE
			faktor := UDINT#1;
		END_IF;
		init := TRUE;
	END_IF;

	IF mode THEN
		T_PLC_MS := DINT_TO_UDINT(PLC_SYS_TICK_CNT) / faktor;
	ELSE
		T_PLC_MS := DINT_TO_UDINT(PLC_SYS_TICK_CNT) * faktor;
	END_IF;

	IF debug THEN
		T_PLC_MS := (DWORD_TO_UDINT(SHL(UDINT_TO_DWORD(T_PLC_MS),N) OR SHL(temp,N)) - UDINT#1) + Offset;
	END_IF;

END_FUNCTION_BLOCK

FUNCTION DT_TO_TOD2:UDINT
	VAR_INPUT
		IN :	UDINT;
	END_VAR

	DT_TO_TOD2 := (IN MOD UDINT#86400) * UDINT#1000;
END_FUNCTION

FUNCTION _DT_TO_DATE_B:UDINT

	VAR_INPUT
		_INN :	UDINT;
	END_VAR

	_DT_TO_DATE_B := (_INN / UDINT#86400) * UDINT#86400;
END_FUNCTION

FUNCTION DAY_OF_WEEK:INT
  VAR_INPUT
    IDATE :	UDINT;
  END_VAR

  DAY_OF_WEEK := UDINT_TO_INT((idate / UDINT#86400 + UDINT#3) MOD UDINT#7) + INT#01;
END_FUNCTION

FUNCTION TIME_TO_UDINT2:UDINT
	VAR_INPUT
		X :	TIME;
	END_VAR

	TIME_TO_UDINT2 := DINT_TO_UDINT(TIME_TO_DINT(X));
END_FUNCTION

FUNCTION_BLOCK TIMER_EXT_Block

	VAR_INPUT
		ENA :	BOOL;
		_ON :	BOOL;
		OFF :	BOOL;
		MAN :	BOOL;
		SWITCH :	BOOL;
		DT_IN :	UDINT;
		SUN_SET :	UDINT;
		SUN_RISE :	UDINT;
		HOLIDAY :	BOOL;
		T_DEBOUNCE :	TIME := T#100ms;
		T_RISE_START :	TIME;
		T_RISE_STOP :	TIME;
		T_SET_START :	TIME;
		T_SET_STOP :	TIME;
		T_DAY_START :	UDINT;
		T_DAY_STOP :	UDINT;
		ENABLE_SATURDAY :	BOOL;
		ENABLE_SUNDAY :	BOOL;
		ENABLE_HOLIDAY :	BOOL;
	END_VAR

	VAR_OUTPUT
		Q :	BOOL;
		STATUS :	BYTE;
	END_VAR

	VAR
		mx :	MANUAL_2_Block;
		deb :	DEBOUNCE_Block;
		tdx :	UDINT;
		wdx :	INT;
		tc :	TIME;
		tx :	UDINT;
		tl :	UDINT;
		qx :	BOOL;
		T_PLC_MS :	T_PLC_MS_Block;
		init :	BOOL;
	END_VAR

	SUN_RISE := SUN_RISE / UDINT#1000 * UDINT#1000;
	SUN_SET := SUN_SET / UDINT#1000 * UDINT#1000;

	T_PLC_MS();
	tx:= T_PLC_MS.T_PLC_MS;
	IF NOT init THEN
		init := TRUE;
		tl := tx;
	END_IF;
	tc := UDINT_TO_TIME(tx - tl);
	IF tc < t#200ms THEN RETURN; END_IF;
	tl := tx;

	deb(in := SWITCH, TD := T_DEBOUNCE, PM := TRUE);

	tdx := DT_TO_TOD2(dt_in);
	wdx := DAY_OF_WEEK(_DT_TO_DATE_B(dt_in));

	IF deb.Q THEN
		qx := NOT qx;
		status := BYTE#110;
	ELSIF holiday AND NOT enable_holiday THEN
		qx := FALSE;
	ELSIF wdx = 6 AND NOT enable_saturday THEN
		qx := FALSE;
	ELSIF wdx = 7 AND NOT enable_sunday THEN
		qx := FALSE;
	ELSIF T_day_start > UDINT#00 AND tdx - T_DAY_START <= TIME_TO_UDINT2(tc) THEN
		qx := TRUE;
		status := BYTE#111;
	ELSIF T_DAY_STOP > UDINT#00 AND tdx - T_DAY_STOP <= TIME_TO_UDINT2(tc) THEN
		qx := FALSE;
		status := BYTE#112;
	ELSIF T_RISE_START > T#0s AND tdx - SUN_RISE + TIME_TO_UDINT2(T_RISE_START) <= TIME_TO_UDINT2(tc) THEN
		qx := TRUE;
		status := BYTE#113;
	ELSIF T_RISE_STOP > T#0s AND tdx - SUN_RISE - TIME_TO_UDINT2(T_RISE_STOP) <= TIME_TO_UDINT2(tc) THEN
		qx := FALSE;
		status := BYTE#114;
	ELSIF T_SET_start > T#0s AND tdx - SUN_SET + TIME_TO_UDINT2(T_SET_START) <= TIME_TO_UDINT2(tc) THEN
		qx := TRUE;
		status := BYTE#115;
	ELSIF T_SET_STOP > T#0s AND tdx - SUN_SET - TIME_TO_UDINT2(T_SET_STOP) <= TIME_TO_UDINT2(tc) THEN
		qx := FALSE;
		status := BYTE#116;
	END_IF;

	mx(_IN := qx, ena := ENA, _ON := _ON, off := OFF, man := MAN);
	Q := mx.Q;

	IF mx.STATUS > BYTE#100 THEN status := mx.STATUS; END_IF;

END_FUNCTION_BLOCK

PROGRAM program0
	VAR
		ENA :	BOOL;
		_ON :	BOOL;
		OFF :	BOOL;
		MAN :	BOOL;
		SWITCH :	BOOL;
		DT_IN :	UDINT;
		SUN_SET :	UDINT;
		SUN_RISE :	UDINT;
		HOLIDAY :	BOOL;
		T_DEBOUNCE :	TIME := T#100ms;
		T_RISE_START :	TIME;
		T_RISE_STOP :	TIME;
		T_SET_START :	TIME;
		T_SET_STOP :	TIME;
		T_DAY_START :	UDINT;
		T_DAY_STOP :	UDINT;
		ENABLE_SATURDAY :	BOOL;
		ENABLE_SUNDAY :	BOOL;
		ENABLE_HOLIDAY :	BOOL;
		Q :	BOOL;
		STATUS :	BYTE;

		func_block : TIMER_EXT_Block;
	END_VAR
	func_block.ENA := ENA;
	func_block._ON := _ON;
	func_block.OFF := OFF ;
	func_block.MAN    := MAN    ;
	func_block.SWITCH := SWITCH;
	func_block.DT_IN := DT_IN;
	func_block.SUN_SET := SUN_SET;
	func_block.SUN_RISE := SUN_RISE ;
	func_block.HOLIDAY    := HOLIDAY    ;
	func_block.T_DEBOUNCE := T_DEBOUNCE;
	func_block.T_RISE_START := T_RISE_START;
	func_block.T_RISE_STOP := T_RISE_STOP;
	func_block.T_SET_START := T_SET_START ;
	func_block.T_SET_STOP    := T_SET_STOP    ;
	func_block.T_DAY_START := T_DAY_START;
	func_block.T_DAY_STOP := T_DAY_STOP;
	func_block.ENABLE_SATURDAY := ENABLE_SATURDAY;
	func_block.ENABLE_SUNDAY := ENABLE_SUNDAY ;
	func_block.ENABLE_HOLIDAY    := ENABLE_HOLIDAY    ;

	func_block();
	Q  := func_block.Q;
	STATUS := func_block.STATUS;
END_PROGRAM

CONFIGURATION Config0
	VAR_GLOBAL
		PLC_TICKS_PER_SEC :	INT;
		PLC_SYS_TICK_CNT :	DINT;
	END_VAR
  	RESOURCE Res0 ON PLC
    	TASK task0(INTERVAL := T#20ms,PRIORITY := 0);
    	PROGRAM instance0 WITH task0 : program0;
  	END_RESOURCE
END_CONFIGURATION

(* ---- TMAX.ST ---- *)
FUNCTION UDINT_TO_TIME2:TIME

	VAR_INPUT
		IN :	UDINT;
	END_VAR

	UDINT_TO_TIME2 := DINT_TO_TIME(UDINT_TO_DINT(IN));

END_FUNCTION

FUNCTION_BLOCK T_PLC_MS_block
	VAR_OUTPUT
		T_PLC_MS :	UDINT;
	END_VAR

	VAR_EXTERNAL
		PLC_TICKS_PER_SEC :	INT;
		PLC_SYS_TICK_CNT :	DINT;
	END_VAR

	VAR
		debug :	BOOL;(*Debug-Mode ON / OFF*)
		N :	INT;(*Debug-Faktor*)
		Offset :	UDINT;(*Debug-Offset*)
		temp :	DWORD := DWORD#1;(*Debug-Offset*)
		mode :	BOOL;(*modus*)
		faktor :	UDINT;(*Systemtakt-Faktor*)
		init :	BOOL;
		v_plc_ticks_per_sec :	UDINT;
		base :	UDINT := UDINT#1000;
	END_VAR

	IF init = FALSE THEN
		v_plc_ticks_per_sec := INT_TO_UDINT(PLC_TICKS_PER_SEC);
		IF v_plc_ticks_per_sec = UDINT#1024 THEN
			faktor := UDINT#1;
			mode := FALSE;
		ELSIF v_plc_ticks_per_sec > UDINT#0 THEN
			IF v_plc_ticks_per_sec <= base THEN
				faktor := base / v_plc_ticks_per_sec;
				mode := FALSE;
			ELSE
				faktor := v_plc_ticks_per_sec / base;
				mode := TRUE;
			END_IF;
		ELSE
			faktor := UDINT#1;
		END_IF;
		init := TRUE;
	END_IF;

	IF mode THEN
		T_PLC_MS := DINT_TO_UDINT(PLC_SYS_TICK_CNT) / faktor;
	ELSE
		T_PLC_MS := DINT_TO_UDINT(PLC_SYS_TICK_CNT) * faktor;
	END_IF;

	IF debug THEN
		T_PLC_MS := (DWORD_TO_UDINT(SHL(UDINT_TO_DWORD(T_PLC_MS),N) OR SHL(temp,N)) - UDINT#1) + Offset;
	END_IF;

END_FUNCTION_BLOCK

FUNCTION_BLOCK TMAX

	VAR_INPUT
		IN :	BOOL;
		PT :	TIME;
	END_VAR

	VAR_OUTPUT
		Q :	BOOL;
		Z :	BOOL;
	END_VAR

	VAR
		tx :	TIME;
		start :	TIME;
		last_in :	BOOL;
		T_PLC_MS :	T_PLC_MS_block;
	END_VAR

	T_PLC_MS();
	tx:= UDINT_TO_TIME(T_PLC_MS.T_PLC_MS);

	Z := FALSE;

	IF NOT in THEN
		Q := FALSE;
	ELSIF IN AND NOT last_in THEN
		Q := TRUE;
		start := tx;
	ELSIF (tx - start >= PT) AND Q THEN
		Q := FALSE;
		Z := TRUE;
	END_IF;

	last_in := IN;

END_FUNCTION_BLOCK

PROGRAM program0
  VAR
	IN :	BOOL;
	PT :	TIME;
	Q :	BOOL;
	Z :	BOOL;
	func_block : TMAX;
  END_VAR
	func_block.IN  :=IN;
	func_block.PT  :=PT;
	func_block();
	Q := func_block.Q;
	Z := func_block.Z;

END_PROGRAM

CONFIGURATION Config0
	VAR_GLOBAL
		PLC_TICKS_PER_SEC :	INT;
		PLC_SYS_TICK_CNT :	DINT;
	END_VAR
	RESOURCE Res0 ON PLC
		TASK task0(INTERVAL := T#20ms,PRIORITY := 0);
		PROGRAM instance0 WITH task0 : program0;
	END_RESOURCE
END_CONFIGURATION

(* ---- TMIN.ST ---- *)
FUNCTION_BLOCK TMIN

	VAR_INPUT
		IN :	BOOL;
		PT :	TIME;
	END_VAR

	VAR_OUTPUT
		Q :	BOOL;
	END_VAR

	VAR
		pm :	TP;
	END_VAR

	pm(in := IN, PT := PT);
	Q := IN OR pm.Q;

END_FUNCTION_BLOCK

PROGRAM program0
  VAR
	IN :	BOOL;
	PT :	TIME;
	Q :	BOOL;
	func_block : TMIN;
  END_VAR
	func_block.IN  :=IN;
	func_block.PT  :=PT;
	func_block();
	Q := func_block.Q;

END_PROGRAM

CONFIGURATION Config0
	RESOURCE Res0 ON PLC
		TASK task0(INTERVAL := T#20ms,PRIORITY := 0);
		PROGRAM instance0 WITH task0 : program0;
	END_RESOURCE
END_CONFIGURATION

(* ---- TN_RECEIVE.ST ---- *)
TYPE
  bya_TN_CHAR:       	ARRAY [0..1919] OF BYTE;
  bya_TN_BACKUP:     	ARRAY [0..1919] OF BYTE;
  bya_TN_COLOR:      	ARRAY [0..1919] OF BYTE;
  bya_TN_Line_Update:	ARRAY [0..23]   OF BOOL;

  us_TN_SCREEN :
  STRUCT
		bya_CHAR:			bya_TN_CHAR;
		bya_COLOR:			bya_TN_COLOR;
		bya_BACKUP:			bya_TN_BACKUP;
		bya_Line_Update:	bya_TN_Line_Update;

		by_Input_Exten_Code:    BYTE;
		by_Input_ASCII_Code:    BYTE;
		bo_Input_ASCII_IsNum:   BOOL;
		in_Page_Number:        	INT;
		in_Cursor_X:           	INT;
		in_Cursor_Y:           	INT;
		in_EOS_Offset:         	INT;
		by_Clear_Screen_Attr:  	BYTE;
		bo_Clear_Screen:       	BOOL;
		bo_Modal_Dialog:       	BOOL;
		bo_Menue_Bar_Dialog:   	BOOL;

  END_STRUCT;
END_TYPE

TYPE
  oscat_NW_BUF_LONG  : ARRAY [0..4095] OF BYTE;

  oscat_NETWORK_BUFFER :
  STRUCT
    SIZE   : UINT;
    BUFFER : oscat_NW_BUF_LONG;
  END_STRUCT;
END_TYPE

FUNCTION ISC_NUM:BOOL

	VAR_INPUT
		IN :	BYTE;
	END_VAR

	ISC_NUM := IN > BYTE#47 AND IN < BYTE#58;

END_FUNCTION

FUNCTION_BLOCK TN_RECEIVE_Block

  VAR_IN_OUT
    R_BUF :	oscat_NETWORK_BUFFER;
    Xus_TN_SCREEN :	us_TN_SCREEN;
  END_VAR

  VAR
    REQ_Size :	UINT;
    REQ1 :	BYTE;
    REQ2 :	BYTE;
    REQ3 :	BYTE;
  END_VAR

  Xus_TN_SCREEN.by_Input_ASCII_Code := BYTE#00;
  Xus_TN_SCREEN.by_Input_Exten_Code := BYTE#00;

  IF R_BUF.SIZE > UINT#0 THEN
    REQ_Size := R_BUF.SIZE;
    REQ1 := R_BUF.BUFFER[0];
    REQ2 := R_BUF.BUFFER[1];
    REQ3 := R_BUF.BUFFER[2];

    IF REQ1 = BYTE#27 AND REQ_Size >= UINT#3 THEN
      IF REQ2 = BYTE#91 THEN
        IF (REQ3 >= BYTE#65 AND REQ3 <= BYTE#68) OR (REQ3 = BYTE#72) OR (REQ3 = BYTE#75) THEN
          Xus_TN_SCREEN.by_Input_Exten_Code := REQ3;
        END_IF;
      ELSIF REQ2 = BYTE#79 THEN
        IF REQ3 >= BYTE#80 AND REQ3 <= BYTE#83 THEN
          Xus_TN_SCREEN.by_Input_Exten_Code := REQ3;
        END_IF;
      END_IF;
    ELSIF REQ1 >= BYTE#32 AND REQ1 <= BYTE#126 THEN
    Xus_TN_SCREEN.by_Input_ASCII_Code := REQ1;
      Xus_TN_SCREEN.bo_Input_ASCII_IsNum := ISC_NUM(REQ1);
    ELSIF REQ1 = BYTE#8 OR REQ1 = BYTE#9 OR REQ1 = BYTE#13 OR REQ1 = BYTE#27 THEN
    Xus_TN_SCREEN.by_Input_Exten_Code := REQ1;
    END_IF;

    R_BUF.SIZE := UINT#00;
  END_IF;

END_FUNCTION_BLOCK

PROGRAM program0
	VAR
		R_BUF :	oscat_NETWORK_BUFFER;
    Xus_TN_SCREEN :	us_TN_SCREEN;

		func_block : TN_RECEIVE_Block;
	END_VAR
	func_block.R_BUF := R_BUF;
	func_block.Xus_TN_SCREEN := Xus_TN_SCREEN;

	func_block();
  R_BUF  := func_block.R_BUF;
	Xus_TN_SCREEN  := func_block.Xus_TN_SCREEN;
END_PROGRAM

CONFIGURATION Config0
	RESOURCE Res0 ON PLC
		TASK task0(INTERVAL := T#20ms,PRIORITY := 0);
		PROGRAM instance0 WITH task0 : program0;
	END_RESOURCE
END_CONFIGURATION

(* ---- TN_SC_AREA_SAVE.ST ---- *)
TYPE
  bya_TN_CHAR:       	ARRAY [0..1919] OF BYTE;
  bya_TN_BACKUP:     	ARRAY [0..1919] OF BYTE;
  bya_TN_COLOR:      	ARRAY [0..1919] OF BYTE;
  bya_TN_Line_Update:	ARRAY [0..23]   OF BOOL;

  us_TN_SCREEN :
  STRUCT
		bya_CHAR:			bya_TN_CHAR;
		bya_COLOR:			bya_TN_COLOR;
		bya_BACKUP:			bya_TN_BACKUP;
		bya_Line_Update:	bya_TN_Line_Update;

		by_Input_Exten_Code:    BYTE;
		by_Input_ASCII_Code:    BYTE;
		bo_Input_ASCII_IsNum:   BOOL;
		in_Page_Number:        	INT;                (* aktive Seiten-Nr.              *)
		in_Cursor_X:           	INT;                (* Cursor X-Position              *)
		in_Cursor_Y:           	INT;                (* Cursor Y-Position              *)
		in_EOS_Offset:         	INT;                (* End of String Offset           *)
		by_Clear_Screen_Attr:  	BYTE;               (* Clear-Screen Attr              *)
		bo_Clear_Screen:       	BOOL;               (* Clear-Screen ausl�sen          *)
		bo_Modal_Dialog:       	BOOL;               (* Modaler Dialog ist aktiv       *)
		bo_Menue_Bar_Dialog:   	BOOL;               (* Menue Dialog ist aktiv         *)

  END_STRUCT;
END_TYPE

FUNCTION TN_SC_XY2_ERROR:BOOL

	VAR_INPUT
		X1 :	INT;
		Y1 :	INT;
		X2 :	INT;
		Y2 :	INT;
	END_VAR

	TN_SC_XY2_ERROR := Y1 < 0 OR X1 < 0 OR Y2 < 0 OR X2 < 0 OR Y1 > 23 OR X1 > 79 OR Y2 > 23 OR X2 > 79;

END_FUNCTION

FUNCTION_BLOCK TN_SC_AREA_SAVE_Block

	VAR
		in_Offset_1 :	INT;
		in_Offset_2 :	INT;
		in_Y :	INT;
		in_X :	INT;
	END_VAR

	VAR_INPUT
		Iin_Y1 :	INT;
		Iin_X1 :	INT;
		Iin_Y2 :	INT;
		Iin_X2 :	INT;
	END_VAR

	VAR_IN_OUT
		Xus_TN_SCREEN :	us_TN_SCREEN;
	END_VAR

	IF TN_SC_XY2_ERROR(Iin_X1,Iin_Y1,Iin_X2,Iin_Y2) THEN RETURN; END_IF;

	Xus_TN_SCREEN.bya_BACKUP[0] := BYTE#1;
	Xus_TN_SCREEN.bya_BACKUP[1] := INT_TO_BYTE(Iin_X1);
	Xus_TN_SCREEN.bya_BACKUP[2] := INT_TO_BYTE(Iin_Y1);
	Xus_TN_SCREEN.bya_BACKUP[3] := INT_TO_BYTE(Iin_X2);
	Xus_TN_SCREEN.bya_BACKUP[4] := INT_TO_BYTE(Iin_Y2);

	in_Offset_2 := 5;
	FOR in_Y := Iin_Y1 TO Iin_Y2 DO

	in_Offset_1 := (in_Y * 80) + Iin_X1;
	FOR in_X := Iin_X1 TO Iin_X2 DO

		Xus_TN_SCREEN.bya_BACKUP[in_Offset_2] := Xus_TN_SCREEN.bya_CHAR[in_Offset_1];
		in_Offset_2 := in_Offset_2 + INT#01;
		Xus_TN_SCREEN.bya_BACKUP[in_Offset_2] := Xus_TN_SCREEN.bya_COLOR[in_Offset_1];
		in_Offset_2 := in_Offset_2 + INT#01;
		in_Offset_1 := in_Offset_1 + INT#01;

	END_FOR;
	END_FOR;

END_FUNCTION_BLOCK

PROGRAM program0
	VAR
		Iin_Y1 :	INT;
		Iin_X1 :	INT;
		Iin_Y2 :	INT;
		Iin_X2 :	INT;
		Xus_TN_SCREEN :	us_TN_SCREEN;

		func_block : TN_SC_AREA_SAVE_Block;
	END_VAR
	func_block.Iin_X1 := Iin_X1;
	func_block.Iin_Y1 := Iin_Y1;
	func_block.Iin_X2 := Iin_X2;
	func_block.Iin_Y2 := Iin_Y2;
	func_block.Xus_TN_SCREEN := Xus_TN_SCREEN;

	func_block();
	Xus_TN_SCREEN  := func_block.Xus_TN_SCREEN;
END_PROGRAM

CONFIGURATION Config0
	RESOURCE Res0 ON PLC
		TASK task0(INTERVAL := T#20ms,PRIORITY := 0);
		PROGRAM instance0 WITH task0 : program0;
	END_RESOURCE
END_CONFIGURATION

(* ---- TN_SC_FILL.ST ---- *)
TYPE
  bya_TN_CHAR:       	ARRAY [0..1919] OF BYTE;
  bya_TN_BACKUP:     	ARRAY [0..1919] OF BYTE;
  bya_TN_COLOR:      	ARRAY [0..1919] OF BYTE;
  bya_TN_Line_Update:	ARRAY [0..23]   OF BOOL;

  us_TN_SCREEN :
  STRUCT
		bya_CHAR:			bya_TN_CHAR;
		bya_COLOR:			bya_TN_COLOR;
		bya_BACKUP:			bya_TN_BACKUP;
		bya_Line_Update:	bya_TN_Line_Update;

		by_Input_Exten_Code:    BYTE;
		by_Input_ASCII_Code:    BYTE;
		bo_Input_ASCII_IsNum:   BOOL;
		in_Page_Number:        	INT;                (* aktive Seiten-Nr.              *)
		in_Cursor_X:           	INT;                (* Cursor X-Position              *)
		in_Cursor_Y:           	INT;                (* Cursor Y-Position              *)
		in_EOS_Offset:         	INT;                (* End of String Offset           *)
		by_Clear_Screen_Attr:  	BYTE;               (* Clear-Screen Attr              *)
		bo_Clear_Screen:       	BOOL;               (* Clear-Screen ausl�sen          *)
		bo_Modal_Dialog:       	BOOL;               (* Modaler Dialog ist aktiv       *)
		bo_Menue_Bar_Dialog:   	BOOL;               (* Menue Dialog ist aktiv         *)

  END_STRUCT;
END_TYPE

FUNCTION TN_SC_XY2_ERROR:BOOL

	VAR_INPUT
		X1 :	INT;
		Y1 :	INT;
		X2 :	INT;
		Y2 :	INT;
	END_VAR

	TN_SC_XY2_ERROR := Y1 < 0 OR X1 < 0 OR Y2 < 0 OR X2 < 0 OR Y1 > 23 OR X1 > 79 OR Y2 > 23 OR X2 > 79;

END_FUNCTION

FUNCTION_BLOCK TN_SC_FILL_Block

	VAR
		in_X :	INT;
		in_Y :	INT;
		in_Offset :	INT;
	END_VAR

	VAR_INPUT
		Iin_Y1 :	INT;
		Iin_X1 :	INT;
		Iin_Y2 :	INT;
		Iin_X2 :	INT;
		Iby_CHAR :	BYTE;
		Iby_Attr :	BYTE;
	END_VAR

	VAR_IN_OUT
		Xus_TN_SCREEN :	us_TN_SCREEN;
	END_VAR

	IF TN_SC_XY2_ERROR(Iin_X1,Iin_Y1,Iin_X2,Iin_Y2) THEN RETURN; END_IF;

	FOR in_Y := Iin_Y1 TO Iin_Y2 DO
	Xus_TN_SCREEN.bya_Line_Update[in_Y] := TRUE;
	in_Offset := (in_Y * 80) + Iin_X1;
	FOR in_X := Iin_X1 TO Iin_X2 DO
		Xus_TN_SCREEN.bya_CHAR[in_Offset]  := Iby_CHAR;
		Xus_TN_SCREEN.bya_COLOR[in_Offset] := Iby_Attr;
		in_Offset := in_Offset + 1;
	END_FOR;
	END_FOR;

END_FUNCTION_BLOCK

PROGRAM program0
	VAR
		Iin_Y1 :	INT;
		Iin_X1 :	INT;
		Iin_Y2 :	INT;
		Iin_X2 :	INT;
		Iby_CHAR :	BYTE;
		Iby_Attr :	BYTE;
		Xus_TN_SCREEN :	us_TN_SCREEN;

		func_block : TN_SC_FILL_Block;
	END_VAR
	func_block.Iin_X1 := Iin_X1;
	func_block.Iin_Y1 := Iin_Y1;
  	func_block.Iin_X2 := Iin_X2;
	func_block.Iin_Y2 := Iin_Y2;
  	func_block.Iby_CHAR := Iby_CHAR;
	func_block.Iby_Attr := Iby_Attr;
	func_block.Xus_TN_SCREEN := Xus_TN_SCREEN;

	func_block();
	Xus_TN_SCREEN  := func_block.Xus_TN_SCREEN;
END_PROGRAM

CONFIGURATION Config0
	RESOURCE Res0 ON PLC
		TASK task0(INTERVAL := T#20ms,PRIORITY := 0);
		PROGRAM instance0 WITH task0 : program0;
	END_RESOURCE
END_CONFIGURATION

(* ---- TN_SC_READ_ATTR.ST ---- *)
TYPE
  bya_TN_CHAR:       	ARRAY [0..1919] OF BYTE;
  bya_TN_BACKUP:     	ARRAY [0..1919] OF BYTE;
  bya_TN_COLOR:      	ARRAY [0..1919] OF BYTE;
  bya_TN_Line_Update:	ARRAY [0..23]   OF BOOL;

  us_TN_SCREEN :
  STRUCT
		bya_CHAR:			bya_TN_CHAR;
		bya_COLOR:			bya_TN_COLOR;
		bya_BACKUP:			bya_TN_BACKUP;
		bya_Line_Update:	bya_TN_Line_Update;

		by_Input_Exten_Code:    BYTE;
		by_Input_ASCII_Code:    BYTE;
		bo_Input_ASCII_IsNum:   BOOL;
		in_Page_Number:        	INT;                (* aktive Seiten-Nr.              *)
		in_Cursor_X:           	INT;                (* Cursor X-Position              *)
		in_Cursor_Y:           	INT;                (* Cursor Y-Position              *)
		in_EOS_Offset:         	INT;                (* End of String Offset           *)
		by_Clear_Screen_Attr:  	BYTE;               (* Clear-Screen Attr              *)
		bo_Clear_Screen:       	BOOL;               (* Clear-Screen ausl�sen          *)
		bo_Modal_Dialog:       	BOOL;               (* Modaler Dialog ist aktiv       *)
		bo_Menue_Bar_Dialog:   	BOOL;               (* Menue Dialog ist aktiv         *)

  END_STRUCT;
END_TYPE

FUNCTION TN_SC_XY_ERROR:BOOL

	VAR_INPUT
		X :	INT;
		Y :	INT;
	END_VAR

	TN_SC_XY_ERROR := Y < 0 OR X < 0 OR Y > 23 OR X > 79;

END_FUNCTION

FUNCTION_BLOCK TN_SC_READ_ATTR_Block

	VAR
		in_Offset :	INT;
	END_VAR

	VAR_INPUT
		Iin_Y :	INT;
		Iin_X :	INT;
	END_VAR

	VAR_OUTPUT
		Oby_ATTR :	BYTE;
	END_VAR

	VAR_IN_OUT
		Xus_TN_SCREEN :	us_TN_SCREEN;
	END_VAR

	IF TN_SC_XY_ERROR(Iin_X,Iin_Y) THEN RETURN; END_IF;
	in_Offset := (Iin_Y * 80) + Iin_X;
	Oby_ATTR := Xus_TN_SCREEN.bya_COLOR[in_Offset];

END_FUNCTION_BLOCK

PROGRAM program0
	VAR
		Iin_Y :	INT;
		Iin_X :	INT;
		Xus_TN_SCREEN :	us_TN_SCREEN;
		Oby_ATTR :	BYTE;

		func_block : TN_SC_READ_ATTR_Block;
	END_VAR
	func_block.Iin_Y := Iin_Y;
	func_block.Iin_X := Iin_X;
	func_block.Xus_TN_SCREEN := Xus_TN_SCREEN;

	func_block();
	Xus_TN_SCREEN  := func_block.Xus_TN_SCREEN;
	Oby_ATTR  := func_block.Oby_ATTR;
END_PROGRAM

CONFIGURATION Config0
	RESOURCE Res0 ON PLC
		TASK task0(INTERVAL := T#20ms,PRIORITY := 0);
		PROGRAM instance0 WITH task0 : program0;
	END_RESOURCE
END_CONFIGURATION

(* ---- TN_SC_READ_CHAR.ST ---- *)
TYPE
  bya_TN_CHAR:       	ARRAY [0..1919] OF BYTE;
  bya_TN_BACKUP:     	ARRAY [0..1919] OF BYTE;
  bya_TN_COLOR:      	ARRAY [0..1919] OF BYTE;
  bya_TN_Line_Update:	ARRAY [0..23]   OF BOOL;

  us_TN_SCREEN :
  STRUCT
		bya_CHAR:			bya_TN_CHAR;
		bya_COLOR:			bya_TN_COLOR;
		bya_BACKUP:			bya_TN_BACKUP;
		bya_Line_Update:	bya_TN_Line_Update;

		by_Input_Exten_Code:    BYTE;
		by_Input_ASCII_Code:    BYTE;
		bo_Input_ASCII_IsNum:   BOOL;
		in_Page_Number:        	INT;                (* aktive Seiten-Nr.              *)
		in_Cursor_X:           	INT;                (* Cursor X-Position              *)
		in_Cursor_Y:           	INT;                (* Cursor Y-Position              *)
		in_EOS_Offset:         	INT;                (* End of String Offset           *)
		by_Clear_Screen_Attr:  	BYTE;               (* Clear-Screen Attr              *)
		bo_Clear_Screen:       	BOOL;               (* Clear-Screen ausl�sen          *)
		bo_Modal_Dialog:       	BOOL;               (* Modaler Dialog ist aktiv       *)
		bo_Menue_Bar_Dialog:   	BOOL;               (* Menue Dialog ist aktiv         *)

  END_STRUCT;
END_TYPE

FUNCTION TN_SC_XY_ERROR:BOOL

	VAR_INPUT
		X :	INT;
		Y :	INT;
	END_VAR

	TN_SC_XY_ERROR := Y < 0 OR X < 0 OR Y > 23 OR X > 79;

END_FUNCTION

FUNCTION_BLOCK TN_SC_READ_CHAR_Block

	VAR
		in_Offset :	INT;
	END_VAR

	VAR_INPUT
		Iin_Y :	INT;
		Iin_X :	INT;
	END_VAR

	VAR_OUTPUT
		Oby_CHAR :	BYTE;
	END_VAR

	VAR_IN_OUT
		Xus_TN_SCREEN :	us_TN_SCREEN;
	END_VAR

	IF TN_SC_XY_ERROR(Iin_X,Iin_Y) THEN RETURN; END_IF;
	in_Offset := (Iin_Y * 80) + Iin_X;
	Oby_CHAR := Xus_TN_SCREEN.bya_CHAR[in_Offset];

END_FUNCTION_BLOCK

PROGRAM program0
	VAR
		Iin_Y :	INT;
		Iin_X :	INT;
		Xus_TN_SCREEN :	us_TN_SCREEN;
		Oby_CHAR :	BYTE;

		func_block : TN_SC_READ_CHAR_Block;
	END_VAR
	func_block.Iin_Y := Iin_Y;
	func_block.Iin_X := Iin_X;
	func_block.Xus_TN_SCREEN := Xus_TN_SCREEN;

	func_block();
	Xus_TN_SCREEN  := func_block.Xus_TN_SCREEN;
	Oby_CHAR  := func_block.Oby_CHAR;
END_PROGRAM

CONFIGURATION Config0
	RESOURCE Res0 ON PLC
		TASK task0(INTERVAL := T#20ms,PRIORITY := 0);
		PROGRAM instance0 WITH task0 : program0;
	END_RESOURCE
END_CONFIGURATION

(* ---- TN_SC_WRITE_ATTR.ST ---- *)
TYPE
  bya_TN_CHAR:       	ARRAY [0..1919] OF BYTE;
  bya_TN_BACKUP:     	ARRAY [0..1919] OF BYTE;
  bya_TN_COLOR:      	ARRAY [0..1919] OF BYTE;
  bya_TN_Line_Update:	ARRAY [0..23]   OF BOOL;

  us_TN_SCREEN :
  STRUCT
		bya_CHAR:			bya_TN_CHAR;
		bya_COLOR:			bya_TN_COLOR;
		bya_BACKUP:			bya_TN_BACKUP;
		bya_Line_Update:	bya_TN_Line_Update;

		by_Input_Exten_Code:    BYTE;
		by_Input_ASCII_Code:    BYTE;
		bo_Input_ASCII_IsNum:   BOOL;
		in_Page_Number:        	INT;                (* aktive Seiten-Nr.              *)
		in_Cursor_X:           	INT;                (* Cursor X-Position              *)
		in_Cursor_Y:           	INT;                (* Cursor Y-Position              *)
		in_EOS_Offset:         	INT;                (* End of String Offset           *)
		by_Clear_Screen_Attr:  	BYTE;               (* Clear-Screen Attr              *)
		bo_Clear_Screen:       	BOOL;               (* Clear-Screen ausl�sen          *)
		bo_Modal_Dialog:       	BOOL;               (* Modaler Dialog ist aktiv       *)
		bo_Menue_Bar_Dialog:   	BOOL;               (* Menue Dialog ist aktiv         *)

  END_STRUCT;
END_TYPE

FUNCTION TN_SC_XY_ERROR:BOOL

	VAR_INPUT
		X :	INT;
		Y :	INT;
	END_VAR

	TN_SC_XY_ERROR := Y < 0 OR X < 0 OR Y > 23 OR X > 79;

END_FUNCTION

FUNCTION_BLOCK TN_SC_WRITE_ATTR_Block

	VAR
		in_Offset :	INT;
	END_VAR

	VAR_INPUT
		Iin_Y :	INT;
		Iin_X :	INT;
		Iby_ATTR :	BYTE;
	END_VAR

	VAR_IN_OUT
		Xus_TN_SCREEN :	us_TN_SCREEN;
	END_VAR

	IF TN_SC_XY_ERROR(Iin_X,Iin_Y) THEN RETURN; END_IF;
	in_Offset := (Iin_Y * 80) + Iin_X;
	Xus_TN_SCREEN.bya_COLOR[in_Offset] := Iby_ATTR;

END_FUNCTION_BLOCK

PROGRAM program0
	VAR
		Iin_Y :	INT;
		Iin_X :	INT;
		Iby_ATTR :	BYTE;
		Xus_TN_SCREEN :	us_TN_SCREEN;

		func_block : TN_SC_WRITE_ATTR_Block;
	END_VAR
	func_block.Iin_Y := Iin_Y;
	func_block.Iin_X := Iin_X;
	func_block.Iby_ATTR := Iby_ATTR;
	func_block.Xus_TN_SCREEN := Xus_TN_SCREEN;

	func_block();
	Xus_TN_SCREEN  := func_block.Xus_TN_SCREEN;
END_PROGRAM

CONFIGURATION Config0
	RESOURCE Res0 ON PLC
		TASK task0(INTERVAL := T#20ms,PRIORITY := 0);
		PROGRAM instance0 WITH task0 : program0;
	END_RESOURCE
END_CONFIGURATION

(* ---- TN_SC_WRITE_CHAR.ST ---- *)
TYPE
  bya_TN_CHAR:       	ARRAY [0..1919] OF BYTE;
  bya_TN_BACKUP:     	ARRAY [0..1919] OF BYTE;
  bya_TN_COLOR:      	ARRAY [0..1919] OF BYTE;
  bya_TN_Line_Update:	ARRAY [0..23]   OF BOOL;

  us_TN_SCREEN :
  STRUCT
		bya_CHAR:			bya_TN_CHAR;
		bya_COLOR:			bya_TN_COLOR;
		bya_BACKUP:			bya_TN_BACKUP;
		bya_Line_Update:	bya_TN_Line_Update;

		by_Input_Exten_Code:    BYTE;
		by_Input_ASCII_Code:    BYTE;
		bo_Input_ASCII_IsNum:   BOOL;
		in_Page_Number:        	INT;                (* aktive Seiten-Nr.              *)
		in_Cursor_X:           	INT;                (* Cursor X-Position              *)
		in_Cursor_Y:           	INT;                (* Cursor Y-Position              *)
		in_EOS_Offset:         	INT;                (* End of String Offset           *)
		by_Clear_Screen_Attr:  	BYTE;               (* Clear-Screen Attr              *)
		bo_Clear_Screen:       	BOOL;               (* Clear-Screen ausl�sen          *)
		bo_Modal_Dialog:       	BOOL;               (* Modaler Dialog ist aktiv       *)
		bo_Menue_Bar_Dialog:   	BOOL;               (* Menue Dialog ist aktiv         *)

  END_STRUCT;
END_TYPE

FUNCTION TN_SC_XY_ERROR:BOOL

	VAR_INPUT
		X :	INT;
		Y :	INT;
	END_VAR

	TN_SC_XY_ERROR := Y < 0 OR X < 0 OR Y > 23 OR X > 79;

END_FUNCTION

FUNCTION_BLOCK TN_SC_WRITE_CHAR_Block

	VAR
		in_Offset :	INT;
	END_VAR

	VAR_INPUT
		Iin_Y :	INT;
		Iin_X :	INT;
		Iby_CHAR :	BYTE;
	END_VAR

	VAR_IN_OUT
		Xus_TN_SCREEN :	us_TN_SCREEN;
	END_VAR

	IF TN_SC_XY_ERROR(Iin_X,Iin_Y) THEN RETURN; END_IF;
	in_Offset := (Iin_Y * 80) + Iin_X;
	Xus_TN_SCREEN.bya_CHAR[in_Offset] := Iby_CHAR;

END_FUNCTION_BLOCK

PROGRAM program0
	VAR
		Iin_Y :	INT;
		Iin_X :	INT;
		Iby_CHAR :	BYTE;
		Xus_TN_SCREEN :	us_TN_SCREEN;

		func_block : TN_SC_WRITE_CHAR_Block;
	END_VAR
	func_block.Iin_Y := Iin_Y;
	func_block.Iin_X := Iin_X;
	func_block.Iby_CHAR := Iby_CHAR;
	func_block.Xus_TN_SCREEN := Xus_TN_SCREEN;

	func_block();
	Xus_TN_SCREEN  := func_block.Xus_TN_SCREEN;
END_PROGRAM

CONFIGURATION Config0
	RESOURCE Res0 ON PLC
		TASK task0(INTERVAL := T#20ms,PRIORITY := 0);
		PROGRAM instance0 WITH task0 : program0;
	END_RESOURCE
END_CONFIGURATION
